(* CoDeSys 2.3 library: TcDrive.lib *)
(* Libraries: STANDARD.LIB 5.6.98 12:03:02, TcBase.lib 14.5.09 12:14:08, TcSystem.lib*7.6.16 10:01:20, TcUtilities.lib*3.2.16 15:08:58, TcEtherCAT.lib*30.11.16 15:34:02, TcTestAndSet.lib 23.2.09 12:50:08 *)

(* Global variable list: Global_Variables *)
VAR_GLOBAL CONSTANT
	S_0_IDN		: WORD	:= 16#0000;
	S_1_IDN		: WORD	:= 16#1000;
	S_2_IDN		: WORD	:= 16#2000;
	S_3_IDN		: WORD	:= 16#3000;
	S_4_IDN		: WORD	:= 16#4000;
	S_5_IDN		: WORD	:= 16#5000;
	S_6_IDN		: WORD	:= 16#6000;
	S_7_IDN		: WORD	:= 16#7000;

	P_0_IDN		: WORD	:= 16#8000;
	P_1_IDN		: WORD	:= 16#9000;
	P_2_IDN		: WORD	:= 16#A000;
	P_3_IDN		: WORD	:= 16#B000;
	P_4_IDN		: WORD	:= 16#C000;
	P_5_IDN		: WORD	:= 16#D000;
	P_6_IDN		: WORD	:= 16#E000;
	P_7_IDN		: WORD	:= 16#F000;
END_VAR
{library private}
VAR_GLOBAL CONSTANT
	iMaxNumOfDrivesUpdate 	: INT := 255;
END_VAR
VAR_GLOBAL
	bBlockEcatScan	 		: BOOL;
	iBlockEcatScanCount		: DINT;
	bBlockDrivesFwUpdate	: BOOL;
	iArrDrivesUpdatePorts 	: ARRAY [0..iMaxNumOfDrivesUpdate] OF UINT;
END_VAR

(* Data type *)
TYPE E_AX5000_DriveOpMode : (
	eOPM_NoModeOfOperation 	:= 0,
	eOPM_TorqueCtrl			:= 1,
	eOPM_VeloCtrl 			:= 2,
	eOPM_PosCtrlFbk1 		:= 3,
	eOPM_PosCtrlFbk2 		:= 4,
	eOPM_PosCtrlFbk1LagLess := 11,
	eOPM_PosCtrlFbk2LagLess := 12
);
END_TYPE

(* Data type *)
TYPE E_FwUpdateState : (
	(* update states *)
	eFwU_NoError := 0,
	eFwU_CheckCfgIdentity,
	eFwU_CheckSlaveCount,
	eFwU_CheckFindSlavePos,
	eFwU_WaitForScan,
	eFwU_ScanningSlaves,
	eFwU_CheckScannedIdentity,
	eFwU_CheckScannedFirmware,
	eFwU_FindFirmwareFile,
	eFwU_WaitForUpdate,
	eFwU_WaitForSlaveState,
	eFwU_StartFwUpdate,
	eFwU_FwUpdateInProgress,
	eFwU_FwUpdateDone,
	eFwU_NoFwUpdateRequired,

	(* not updating via this channel *)
	eFwU_UpdateViaOtherChannelActive,
	eFwU_UpdatedViaOtherChannel,

	(* error states *)
	eFwU_GetSlaveIdentityError			:= -1,
	eFwU_GetSlaveCountError				:= -2,
	eFwU_GetSlaveAddrError				:= -3,
	eFwU_StartScanError					:= -4,
	eFwU_ScanStateError					:= -5,
	eFwU_ScanIdentityError				:= -6,
	eFwU_GetSlaveStateError				:= -7,
	eFwU_ScanFirmwareError				:= -8,
	eFwU_FindFileError					:= -9,
	eFwU_CfgTypeInNoAX5xxx				:= -10,
	eFwU_ScannedTypeInNoAX5xxx			:= -11,
	eFwU_ChannelMismatch				:= -12,
	eFwU_ChannelMismatch_1Cfg_2Scanned	:= -13,
	eFwU_ChannelMismatch_2Cfg_1Scanned	:= -14,
	eFwU_CurrentMismatch				:= -15,
	eFwU_FwUpdateError					:= -16,
	eFwU_ReqSlaveStateError				:= -17,
	eFwU_ChannelMismatch_0Cfg_1Scanned	:= -18,
	eFwU_ChannelMismatch_0Cfg_2Scanned	:= -19,
	eFwU_ChannelMismatch_1Cfg_0Scanned	:= -20,
	eFwU_ChannelMismatch_2Cfg_0Scanned	:= -21,
	eFwU_TypeIncompatibleCfgToScanned	:= -22
);
END_TYPE

(* Data type *)
TYPE E_IndraDriveCs_DriveOpMode : (
	eIDC_NoModeOfOperation := 0,
	eIDC_TorqueCtrl		:= 1,
	eIDC_VeloCtrl 			:= 2,

	eIDC_PosCtrlFbk1 		:= 3,
	eIDC_PosCtrlFbk2 		:= 4,
	eIDC_PosCtrlFbk1LagLess := 11,
	eIDC_PosCtrlFbk2LagLess := 12,

	eIDC_DrvInternInterpolFbk1 := 19,
	eIDC_DrvInternInterpolFbk2 := 20,
	eIDC_DrvInternInterpolFbk1LagLess := 27,
	eIDC_DrvInternInterpolFbk2LagLess := 28,

	eIDC_PosBlockModeFbk1 := 51,
	eIDC_PosBlockModeFbk2 := 52,
	eIDC_PosBlockModeFbk1LagLess := 59,
	eIDC_PosBlockModeFbk2LagLess := 60,

	eIDC_PosCtrlDrvCtrldFbk1 := 259,
	eIDC_PosCtrlDrvCtrldFbk2 := 260,
	eIDC_PosCtrlDrvCtrldFbk1LagLess := 267,
	eIDC_PosCtrlDrvCtrldFbk2LagLess := 268,

	eIDC_DrvCtrldPositioningFbk1 := 531,
	eIDC_DrvCtrldPositioningFbk2 := 532,
	eIDC_DrvCtrldPositioningFbk1LagLess := 539,
	eIDC_DrvCtrldPositioningFbk2LagLess := 540,

	eIDC_CamFbk1VirtMaster := -30717,
	eIDC_CamFbk2VirtMaster := -30716,
	eIDC_CamFbk1VirtMasterLagLess := -30709,
	eIDC_CamFbk2VirtMasterLagLess := -30708,

	eIDC_CamFbk1RealMaster := -30701,
	eIDC_CamFbk2RealMaster := -30700,
	eIDC_CamFbk1RealMasterLagLess := -30693,
	eIDC_CamFbk2RealMasterLagLess := -30692,

	eIDC_PhaseSyncFbk1VirtMaster := -28669,
	eIDC_PhaseSyncFbk2VirtMaster := -28668,
	eIDC_PhaseSyncFbk1VirtMasterLagLess := -28661,
	eIDC_PhaseSyncFbk2VirtMasterLagLess := -28660,

	eIDC_PhaseSyncFbk1RealMaster := -28653,
	eIDC_PhaseSyncFbk2RealMaster := -28652,
	eIDC_PhaseSyncFbk1RealMasterLagLess := -28645,
	eIDC_PhaseSyncFbk2RealMasterLagLess := -28644,

	eIDC_VeloSyncVirtMaster := -24574,
	eIDC_VeloSyncRealMaster := -24558,

	eIDC_MotionProfileFbk1VirtMaster := -26621,
	eIDC_MotionProfileFbk2VirtMaster := -26620,
	eIDC_MotionProfileLagLessFbk1VirtMaster := -26613,
	eIDC_MotionProfileLagLessFbk2VirtMaster := -26612,

	eIDC_MotionProfileFbk1RealMaster := -26605,
	eIDC_MotionProfileFbk2RealMaster := -26604,
	eIDC_MotionProfileLagLessFbk1RealMaster := -26597,
	eIDC_MotionProfileLagLessFbk2RealMaster := -26596,

	eIDC_PosCtrlDrvCtrld := 773,
	eIDC_DrvCtrldPositioning := 533,
	eIDC_PosBlockMode := 565,
	eIDC_VeloSynchronization := 66,
	eIDC_PosSynchronization := 581

);
END_TYPE

(* Data type *)
TYPE E_SoE_AttribLen : (
	eSoE_LEN_2BYTE	:= 1,
	eSoE_LEN_4BYTE	:= 2,
	eSoE_LEN_8BYTE	:= 3,
	eSoE_LEN_V1BYTE	:= 4,
	eSoE_LEN_V2BYTE	:= 5,
	eSoE_LEN_V4BYTE	:= 6,
	eSoE_LEN_V8BYTE	:= 7
);
END_TYPE

(* Data type *)
TYPE E_SoE_CmdControl :(
	eSoE_CmdControl_Cancel				:= 0,
	eSoE_CmdControl_Set					:= 1,
	eSoE_CmdControl_SetAndEnable		:= 3
	);
END_TYPE

(* Data type *)
TYPE E_SoE_CmdState :(
	eSoE_CmdState_NotSet					:= 0,
	eSoE_CmdState_Set						:= 1,
	eSoE_CmdState_Executed					:= 2,
	eSoE_CmdState_SetEnabledExecuted		:= 3,
	eSoE_CmdState_SetAndInterrupted			:= 5,
	eSoE_CmdState_SetEnabledNotExecuted	:= 7,
	eSoE_CmdState_Error						:= 15
);
END_TYPE

(* Data type *)
TYPE E_SoE_Type : (
	eSoE_Type_BIN			:= 0,
	eSoE_Type_UNSIGNED	:= 1,
	eSoE_Type_SIGNED		:= 2,
	eSoE_Type_HEX			:= 3,
	eSoE_Type_TEXT		:= 4,
	eSoE_Type_IDN			:= 5,
	eSoE_Type_FLOAT		:= 6
);
END_TYPE

(* Data type *)
TYPE ST_AX5000_C1D :
STRUCT
	bOverloadShutdown			: BOOL; (* C1D Bit  0 *)
	bAmplifierOverTempShutdown	: BOOL; (* C1D Bit  1 *)
	bMotorOverTempShutdown		: BOOL; (* C1D Bit  2 *)
	bCoolingErrorShutdown		: BOOL; (* C1D Bit  3 *)

	bControlVoltageError		: BOOL; (* C1D Bit  4 *)
	bFeedbackError				: BOOL; (* C1D Bit  5 *)
	bCommunicationError			: BOOL; (* C1D Bit  6 *)
	bOverCurrentError			: BOOL; (* C1D Bit  7 *)

	bOverVoltageError			: BOOL; (* C1D Bit  8 *)
	bUnderVoltageError			: BOOL; (* C1D Bit  9 *)
	bPowerSupplyPhaseError		: BOOL; (* C1D Bit 10 *)
	bExcessivePosDiviationError : BOOL; (* C1D Bit 11 *)

	bCommunicationErrorBit		: BOOL; (* C1D Bit 12 *)
	bOvertravelLimitExceeeded	: BOOL; (* C1D Bit 13 *)
	bReserved 					: BOOL; (* C1D Bit 14 *)
	bManufacturerSpecificError	: BOOL; (* C1D Bit 15 *)
END_STRUCT
END_TYPE

(* Data type *)
TYPE ST_AX5000DriveStatus :
STRUCT
	bStatusCmdValProcessing 	: BOOL;
	bRealTimeStatusBit1 		: BOOL;
	bRealTimeStatusBit2 		: BOOL;
	bDrvShutdownBitC1D		 	: BOOL;
	bChangeBitC2D		 		: BOOL;
	bChangeBitC3D		 		: BOOL;
	bNotReadyToPowerUp			: BOOL;
	bReadyForPower				: BOOL;
	bReadyForEnable				: BOOL;
	bEnabled					: BOOL;
	iActOpModeParNum			: UINT;
	eActOpMode					: E_AX5000_DriveOpMode;
	iReserved					: UINT;
END_STRUCT
END_TYPE

(* Data type *)
TYPE ST_IndraDriveCs_C1D :
STRUCT
	bOverloadShutdown			: BOOL; (* C1D Bit  0 *)
	bAmplifierOverTempShutdown	: BOOL; (* C1D Bit  1 *)
	bMotorOverTempShutdown		: BOOL; (* C1D Bit  2 *)
	bReserved_3					: BOOL; (* C1D Bit  3 *)

	bControlVoltageError		: BOOL; (* C1D Bit  4 *)
	bFeedbackError				: BOOL; (* C1D Bit  5 *)
	bReserved_6					: BOOL; (* C1D Bit  6 *)
	bOverCurrentError			: BOOL; (* C1D Bit  7 *)

	bOverVoltageError			: BOOL; (* C1D Bit  8 *)
	bUnderVoltageError			: BOOL; (* C1D Bit  9 *)
	bReserved_10				: BOOL; (* C1D Bit 10 *)
	bExcessivePosDiviationError : BOOL; (* C1D Bit 11 *)

	bCommunicationErrorBit		: BOOL; (* C1D Bit 12 *)
	bOvertravelLimitExceeeded	: BOOL; (* C1D Bit 13 *)
	bReserved_14				: BOOL; (* C1D Bit 14 *)
	bManufacturerSpecificError	: BOOL; (* C1D Bit 15 *)
END_STRUCT
END_TYPE

(* Data type *)
TYPE ST_IndraDriveCsDriveStatus :
STRUCT
	bStatusCmdValProcessing 	: BOOL;
	bRealTimeStatusBit1 		: BOOL;
	bRealTimeStatusBit2 		: BOOL;
	bDrvShutdownBitC1D		 	: BOOL;
	bChangeBitC2D		 		: BOOL;
	bChangeBitC3D		 		: BOOL;
	bNotReadyToPowerUp			: BOOL;
	bReadyForPower				: BOOL;
	bReadyForEnable				: BOOL;
	bEnabled					: BOOL;
	iActOpModeParNum			: UINT;
	eActOpMode					: E_IndraDriveCs_DriveOpMode;
	iReserved					: UINT;
END_STRUCT
END_TYPE

(* Data type *)
TYPE ST_SoE_CPxInvParamList : ST_SoE_CPxInvParamList25;
END_TYPE

(* Data type *)
TYPE ST_SoE_CPxInvParamList25 :
STRUCT
	iActualSize 	: UINT;
	iMaxSize 		: UINT;
	arrIdnNumbers	: ARRAY [1..25] OF UDINT;
END_STRUCT
END_TYPE

(* Data type *)
TYPE ST_SoE_DiagNumList : ST_SoE_DiagNumList30;
END_TYPE

(* Data type *)
TYPE ST_SoE_DiagNumList30 :
STRUCT
	iActualSize 	: UINT;
	iMaxSize 		: UINT;
	arrDiagNumbers	: ARRAY [0..29] OF UDINT;
END_STRUCT
END_TYPE

(* Data type *)
TYPE ST_SoE_DiagNumList50 :
STRUCT
	iActualSize 	: UINT;
	iMaxSize 		: UINT;
	arrDiagNumbers	: ARRAY [0..49] OF UDINT;
END_STRUCT
END_TYPE

(* Data type *)
TYPE ST_SoE_String :
STRUCT
	iActualSize : UINT;
	iMaxSize 	: UINT;
	strData		: STRING(MAX_STRING_LENGTH);
END_STRUCT
END_TYPE

(* Data type *)
TYPE ST_SoE_StringEx :
STRUCT
	dwAttribute : DWORD;
	iActualSize : UINT;
	iMaxSize 	: UINT;
	strData		: STRING(MAX_STRING_LENGTH);
END_STRUCT
END_TYPE

(* POU F_ConvWordToSTAX5000C1D, ST *)
FUNCTION F_ConvWordToSTAX5000C1D : ST_AX5000_C1D
VAR_INPUT
	wClass1Diag  : WORD;
END_VAR
VAR
	stAX5000C1D	: ST_AX5000_C1D;
END_VAR
stAX5000C1D.bOverloadShutdown			:= wClass1Diag.0;
stAX5000C1D.bAmplifierOverTempShutdown	:= wClass1Diag.1;
stAX5000C1D.bMotorOverTempShutdown		:= wClass1Diag.2;
stAX5000C1D.bCoolingErrorShutdown		:= wClass1Diag.3;

stAX5000C1D.bControlVoltageError		:= wClass1Diag.4;
stAX5000C1D.bFeedbackError				:= wClass1Diag.5;
stAX5000C1D.bCommunicationError			:= wClass1Diag.6;
stAX5000C1D.bOverCurrentError			:= wClass1Diag.7;

stAX5000C1D.bOverVoltageError			:= wClass1Diag.8;
stAX5000C1D.bUnderVoltageError			:= wClass1Diag.9;
stAX5000C1D.bPowerSupplyPhaseError		:= wClass1Diag.10;
stAX5000C1D.bExcessivePosDiviationError := wClass1Diag.11;

stAX5000C1D.bCommunicationErrorBit		:= wClass1Diag.12;
stAX5000C1D.bOvertravelLimitExceeeded	:= wClass1Diag.13;
stAX5000C1D.bReserved 					:= wClass1Diag.14;
stAX5000C1D.bManufacturerSpecificError	:= wClass1Diag.15;

F_ConvWordToSTAX5000C1D := stAX5000C1D;
END_FUNCTION

(* POU F_ConvWordToSTAX5000DriveStatus, ST *)
FUNCTION F_ConvWordToSTAX5000DriveStatus : ST_AX5000DriveStatus
VAR_INPUT
	wDriveStatus  	: WORD;
END_VAR
VAR
	stDriveStatus	: ST_AX5000DriveStatus;
	iOpModeSelect	: INT;
END_VAR
stDriveStatus.bStatusCmdValProcessing := wDriveStatus.3;

stDriveStatus.bRealTimeStatusBit1 := wDriveStatus.6;
stDriveStatus.bRealTimeStatusBit2 := wDriveStatus.7;

iOpModeSelect := 0;
IF wDriveStatus.8 THEN
	iOpModeSelect := iOpModeSelect + 1;
END_IF
IF wDriveStatus.9 THEN
	iOpModeSelect := iOpModeSelect + 2;
END_IF
IF wDriveStatus.10 THEN
	iOpModeSelect := iOpModeSelect + 4;
END_IF

CASE iOpModeSelect OF
0: stDriveStatus.iActOpModeParNum := 32;
1: stDriveStatus.iActOpModeParNum := 33;
2: stDriveStatus.iActOpModeParNum := 34;
3: stDriveStatus.iActOpModeParNum := 35;
4: stDriveStatus.iActOpModeParNum := 284;
5: stDriveStatus.iActOpModeParNum := 285;
6: stDriveStatus.iActOpModeParNum := 286;
7: stDriveStatus.iActOpModeParNum := 287;
END_CASE

stDriveStatus.bChangeBitC3D			:= wDriveStatus.11;
stDriveStatus.bChangeBitC2D			:= wDriveStatus.12;
stDriveStatus.bDrvShutdownBitC1D	:= wDriveStatus.13;

IF wDriveStatus.14 THEN
	IF wDriveStatus.15 THEN (* 3 *)
		stDriveStatus.bNotReadyToPowerUp := FALSE;
		stDriveStatus.bReadyForPower := TRUE;
		stDriveStatus.bReadyForEnable := TRUE;
		stDriveStatus.bEnabled := TRUE;
	ELSE (* 1 *)
		stDriveStatus.bNotReadyToPowerUp := FALSE;
		stDriveStatus.bReadyForPower := TRUE;
		stDriveStatus.bReadyForEnable := FALSE;
		stDriveStatus.bEnabled := FALSE;
	END_IF
ELSE
	IF wDriveStatus.15 THEN (* 2 *)
		stDriveStatus.bNotReadyToPowerUp := FALSE;
		stDriveStatus.bReadyForPower := TRUE;
		stDriveStatus.bReadyForEnable := TRUE;
		stDriveStatus.bEnabled := FALSE;
	ELSE (* 0 *)
		stDriveStatus.bNotReadyToPowerUp := TRUE;
		stDriveStatus.bReadyForPower := FALSE;
		stDriveStatus.bReadyForEnable := FALSE;
		stDriveStatus.bEnabled := FALSE;
	END_IF
END_IF
F_ConvWordToSTAX5000DriveStatus := stDriveStatus;
END_FUNCTION

(* POU F_ConvWordToSTIndraDriveCsC1D, ST *)
FUNCTION F_ConvWordToSTIndraDriveCsC1D : ST_IndraDriveCs_C1D
VAR_INPUT
	wClass1Diag  : WORD;
END_VAR
VAR
	stIndraDriveCsC1D	: ST_IndraDriveCs_C1D;
END_VAR
stIndraDriveCsC1D.bOverloadShutdown				:= wClass1Diag.0;
stIndraDriveCsC1D.bAmplifierOverTempShutdown	:= wClass1Diag.1;
stIndraDriveCsC1D.bMotorOverTempShutdown		:= wClass1Diag.2;
stIndraDriveCsC1D.bReserved_3					:= wClass1Diag.3;

stIndraDriveCsC1D.bControlVoltageError			:= wClass1Diag.4;
stIndraDriveCsC1D.bFeedbackError				:= wClass1Diag.5;
stIndraDriveCsC1D.bReserved_6					:= wClass1Diag.6;
stIndraDriveCsC1D.bOverCurrentError				:= wClass1Diag.7;

stIndraDriveCsC1D.bOverVoltageError				:= wClass1Diag.8;
stIndraDriveCsC1D.bUnderVoltageError			:= wClass1Diag.9;
stIndraDriveCsC1D.bReserved_10					:= wClass1Diag.10;
stIndraDriveCsC1D.bExcessivePosDiviationError 	:= wClass1Diag.11;

stIndraDriveCsC1D.bCommunicationErrorBit		:= wClass1Diag.12;
stIndraDriveCsC1D.bOvertravelLimitExceeeded		:= wClass1Diag.13;
stIndraDriveCsC1D.bReserved_14 					:= wClass1Diag.14;
stIndraDriveCsC1D.bManufacturerSpecificError	:= wClass1Diag.15;

F_ConvWordToSTIndraDriveCsC1D := stIndraDriveCsC1D;
END_FUNCTION

(* POU F_ConvWordToSTIndraDriveCsDriveStatus, ST *)
FUNCTION F_ConvWordToSTIndraDriveCsDriveStatus : ST_IndraDriveCsDriveStatus
VAR_INPUT
	wDriveStatus  	: WORD;
END_VAR
VAR
	stDriveStatus	: ST_IndraDriveCsDriveStatus;
	iOpModeSelect	: INT;
END_VAR
stDriveStatus.bStatusCmdValProcessing := wDriveStatus.3;

stDriveStatus.bRealTimeStatusBit1 := wDriveStatus.6;
stDriveStatus.bRealTimeStatusBit2 := wDriveStatus.7;

iOpModeSelect := 0;
IF wDriveStatus.8 THEN
	iOpModeSelect := iOpModeSelect + 1;
END_IF
IF wDriveStatus.9 THEN
	iOpModeSelect := iOpModeSelect + 2;
END_IF
IF wDriveStatus.10 THEN
	iOpModeSelect := iOpModeSelect + 4;
END_IF

CASE iOpModeSelect OF
0: stDriveStatus.iActOpModeParNum := 32;
1: stDriveStatus.iActOpModeParNum := 33;
2: stDriveStatus.iActOpModeParNum := 34;
3: stDriveStatus.iActOpModeParNum := 35;
4: stDriveStatus.iActOpModeParNum := 284;
5: stDriveStatus.iActOpModeParNum := 285;
6: stDriveStatus.iActOpModeParNum := 286;
7: stDriveStatus.iActOpModeParNum := 287;
END_CASE

stDriveStatus.bChangeBitC3D			:= wDriveStatus.11;
stDriveStatus.bChangeBitC2D			:= wDriveStatus.12;
stDriveStatus.bDrvShutdownBitC1D	:= wDriveStatus.13;

IF wDriveStatus.14 THEN
	IF wDriveStatus.15 THEN (* 3 = AF *)
		stDriveStatus.bNotReadyToPowerUp := FALSE;
		stDriveStatus.bReadyForPower := TRUE;
		stDriveStatus.bReadyForEnable := TRUE;
		stDriveStatus.bEnabled := TRUE;
	ELSE (* 1 = bb *)
		stDriveStatus.bNotReadyToPowerUp := FALSE;
		stDriveStatus.bReadyForPower := TRUE;
		stDriveStatus.bReadyForEnable := FALSE;
		stDriveStatus.bEnabled := FALSE;
	END_IF
ELSE
	IF wDriveStatus.15 THEN (* 2 = AB *)
		stDriveStatus.bNotReadyToPowerUp := FALSE;
		stDriveStatus.bReadyForPower := TRUE;
		stDriveStatus.bReadyForEnable := TRUE;
		stDriveStatus.bEnabled := FALSE;
	ELSE (* 0 = e.g. P2 *)
		stDriveStatus.bNotReadyToPowerUp := TRUE;
		stDriveStatus.bReadyForPower := FALSE;
		stDriveStatus.bReadyForEnable := FALSE;
		stDriveStatus.bEnabled := FALSE;
	END_IF
END_IF
F_ConvWordToSTIndraDriveCsDriveStatus := stDriveStatus;
END_FUNCTION

(* POU F_GetVersionTcDrive, ST *)
FUNCTION F_GetVersionTcDrive : UINT
(* Returns the library version information  *)
VAR_INPUT
	nVersionElement       :       INT;
END_VAR
VAR
END_VAR
(* Version history:
Date          	| Version 	| created under 	     	| Author	| Remark 
------------------------------------------------------------------------------------------------------------------------------------------------------ 
15.05.2008    	| 0.0.1     | V2.10.0 (Build 1325) 		| I.Ch.		| first release 
13.06.2008    	| 0.0.2     | V2.10.0 (Build 1325) 		| I.Ch.		| FB_SoEAX5000Reset_ByDriveRef added
17.06.2008		| 0.0.3		| V2.10.0 (Build 1326)		| AnK		| Don't read the attribute from P-0-0352 in FB_SoEAX5000Reset_ByDriveRef
10.07.2008		| 0.0.4		| V2.10.0 (Build 1326)		| PKa		| FB_SoEAX5000Reset_ByDriveRef, Reset sequence changed PreOP-S.0.0099-OP
11.07.2008		| 0.0.5		| V2.10.0 (Build 1328)		| PKa		| FB_SoEAX5000Reset_ByDriveRef, Read S.0.0011 for DriveError, Reset sequence changed S.0.0099-ClearErrorOP
28.07.2008		| 0.0.6		| V2.10.0 (Build 1328)		| I.Ch.		| using of ST_DriveRef instead of ST_SoE_DriveRef
28.08.2008		| 0.0.7		| V2.10.0 (Build 1328)		| I.Ch.		| FB_SoEAX5000Reset_ByDriveRef removed, FB_SoEReset_ByDriveRef modified
29.09.2008		| 0.0.8		| V2.10.0 (Build 1328)		| I.Ch.		| FB_SoEReset_ByDriveRef: removed check for OP state
02.10.2008		| 0.0.9		| V2.10.0 (Build 1328)		| I.Ch.		| folders added
12.12.2008		| 0.0.10	| V2.10.0 (Build 1330)		| I.Ch.		| FB_SoEAX5000FirmwareUpdate_ByDriveRef added
12.12.2008		| 0.0.11	| V2.10.0 (Build 1330)		| I.Ch.		| TestAndSet semaphore added
13.12.2008		| 0.0.12	| V2.10.0 (Build 1330)		| I.Ch.		| parallel firmware download added
15.12.2008		| 0.0.13	| V2.10.0 (Build 1330)		| I.Ch.		| cleanup
16.12.2008		| 0.0.14	| V2.10.0 (Build 1330)		| I.Ch.		| provide FB_EcFoeLoad.sInfo as iDiagNumber
16.01.2009		| 0.0.15	| V2.10.0 (Build 1331)		| I.Ch.		| provide FirmwareUpdate for >128 EtherCAT Slaves
22.01.2009		| 0.0.16	| V2.11.0 (Build 1513)		| AnK		| FB_SoEAX5000FirmwareUpdate_ByDriveRef: Change file names from AX5200-0000- to AX52xx-xxxx-
03.02.2009		| 0.0.17	| V2.11.0 (Build 1332)		| I.Ch.		| FB_SoEAX5000FirmwareUpdate_ByDriveRef: Change file names AX51/AX52xx-xxxx- to AX5yxx-xxxx-; added AX50**-xxxx
04.02.2009		| 0.0.18	| V2.11.0 (Build 1332)		| I.Ch.		| FB_SoEAX5000FirmwareUpdate_ByDriveRef: fix for filename: '_' instead of '-' (AX5yxx_xxxx_...) 
05.02.2009		| 0.0.19	| V2.11.0 (Build 1332)		| I.Ch.		| cleanup 
15.03.2009		| 0.0.20	| V2.11.0 (Build 1334)		| I.Ch.		| FB_SoEReadClassXDiag_ByDriveRef added, reads C1D|C2D|C3D class diag, F_ConvWordToSTAX5000C1D + ST_AX5000_C1D added 
19.03.2009		| 0.0.21	| V2.11.0 (Build 1334)		| I.Ch.		| Conversion FUs for DriveState/EcSlaveState + DTs DriveState/EcSlaveState, ST_SoE_CPxInvParamList added 
23.03.2009		| 0.0.22	| V2.11.0 (Build 1334)		| I.Ch.		| Conversion FUs for EcSlaveState + EcSlaveState move to TcEtherCAT.lib added 
19.10.2009		| 0.0.23	| V2.11.0 (Build 1539)		| I.Ch.		| optional sequential reading of attribute and value (bSeqReadDrvAttrAndValue) added for other drives than AX5000 in
																		FB_SoEReadClassXDiag_ByDriveRef, FB_SoEReadDiagMessage_ByDriveRef, FB_SoEReadDiagNumber_ByDriveRef, FB_SoEReadAmplifierTemperature_ByDriveRef
																		FB_SoEReadDcBusCurrent_ByDriveRef, FB_SoEReadDcBusVoltage_ByDriveRef, FB_SoEReadMotorTemperature_ByDriveRef
19.10.2009		| 0.0.24	| V2.11.0 (Build 1539)		| I.Ch.		| bSeqReadDrvAttrAndValue moved to TcEtherCAT.lib
13.01.2010		| 0.0.25	| V2.11.0 (Build 1541)		| I.Ch.		| ST_SoE_DiagNumList30, ST_SoE_DiagNumList50 added, ST_SoE_DiagNumList as ALIAS type; ST_SoE_CPxInvParamList25 added, ST_SoE_CPxInvParamList as ALIAS type 
																		Conversion Functions/Datatypes for IndraDriveCs added
17.03.2010		| 0.0.26	| V2.11.0 (Build 1544)		| AnK.		| FB_SoEExecuteCommand_ByDriveRef: Change the handling in case of a command error
02.10.2012		| 0.0.27	| V2.11.0 (Build 1557)		| I.Ch.		| FB_SoEAX5000FirmwareUpdate_ByDriveRef supports FW Update for HW2 in compatible mode (HW1 configured)
24.01.2017		| 0.0.28	| V2.11.0 (Build 2256)		| I.Ch.		| FB_SoEAX5000FirmwareUpdate_ByDriveRef adjusted to also use "_dual_use_conform" firmware files
*)
CASE nVersionElement OF
1: (* major number *)
       F_GetVersionTcDrive := 0;
2: (* minor number *)
       F_GetVersionTcDrive := 0;
3: (* revision number *)
       F_GetVersionTcDrive := 28;
ELSE
   F_GetVersionTcDrive := 16#FFFF;
END_CASE
END_FUNCTION

(* POU FB_SoEAX5000FirmwareUpdate_ByDriveRef, ST *)
FUNCTION_BLOCK FB_SoEAX5000FirmwareUpdate_ByDriveRef
VAR_INPUT
	stDriveRef				: ST_DriveRef; 	(* contains sNetID of EcMaster, nSlaveAddr of EcDrive, nDriveNo of EcDrive, either preset or read from NC *)
	bExecute				: BOOL;			(* Function block execution is triggered by a rising edge at this input.*)
	tTimeout				: TIME := DEFAULT_ADS_TIMEOUT;(* States the time before the function is cancelled. *)
	sFirmwareVersion		: STRING(20);	(* version string vx_yy_bnnnn,
												"v1.05_b0009" 		for specific build: v1.05 Build 0009, 
												"v1.05_b00??" 		for specific version v1.05 latest release build, 
												"v1.??_b00??" 		for latest v1.xx version latest release build
												"v?.??_b00??", "" 	for latest version latest release build 

												"v1.05_b10??" - "v1_05_b89??"  	
																	for specific version v1.05 latest customer specific build, 
												"v1.05_b90??" 		for specific version v1.05 latest debug build, 

												same wildcards for versions 2.xx Build yyyy
												"v2.03_b0026" 		for specific build: v2.03 Build 0026, 
												"v2.03_b00??" 		for specific version v2.03 latest release build, 
												...
											*)
	sFirmwarePath			: T_MaxString;	(* drive:\path, e.g. "C:\TwinCAT\Io\TcDriveManager\FirmwarePool" *)
	sNetIdIPC				: T_AmsNetId;
	iReqEcState				: UINT := EC_DEVICE_STATE_OP;
END_VAR
VAR_OUTPUT
	bBusy					: BOOL;
	bError					: BOOL;
	iAdsErrId				: UINT;
	iSercosErrId			: UINT;
	iDiagNumber				: UDINT;
	eFwUpdateState			: E_FwUpdateState;
	iLoadProgress			: INT;
	sSelectedFirmwareFile	: STRING(MAX_STRING_LENGTH);	(* found firmware file, e.g. "AX5yxx_xxxx_0010_v1_05_b0009.efw" or "AX5yxx_xxxx_0010_v1_05_b0009_dual_use_conform.efw" *)
END_VAR
{library private}
VAR
	iState					: INT;
	bExecute_I				: BOOL;
	iErrId					: UDINT;
	I						: DINT;
	iNextUpdateIdx			: INT;
	iCurUpdateIdx			: INT;
	bUpdateViaOtherChn		: BOOL;

	sConfiguredType 		: STRING(20);	(* type of slave, e.g. "AX5206-0000-0009" *)
	sScannedType 			: STRING(20);	(* type of slave, e.g. "AX5206-0000-0010" *)

	sConfiguredFirmwareFile		: STRING(MAX_STRING_LENGTH);(* configured firmware file, e.g. 	"AX5yxx_xxxx_0010_v1_05_b0003.efw" or "AX5021_xxxx_0009_v1_04_b0002.efw" *)
	sScannedFirmwareFile		: STRING(MAX_STRING_LENGTH);(* scanned firmware file, e.g. 		"AX5yxx_xxxx_0010_v1_05_b0003.efw" or "AX5021_xxxx_0009_v1_04_b0002.efw" *)
	sCompatibleFirmwareFile		: STRING(MAX_STRING_LENGTH);(* compatible firmware file, e.g. 	"AX5yxx_xxxx_0200_v2_03_b0026.efw" or "AX5021_xxxx_0200_v2_03_b0026.efw" *)

	sConfiguredFirmwareFileDUC	: STRING(MAX_STRING_LENGTH);(* configured firmware file, e.g. 	"AX5yxx_xxxx_0010_v1_05_b0003_dual_use_conform.efw" or "AX5021_xxxx_0009_v1_04_b0002_dual_use_conform.efw" *)
	sScannedFirmwareFileDUC		: STRING(MAX_STRING_LENGTH);(* scanned firmware file, e.g. 		"AX5yxx_xxxx_0010_v1_05_b0003_dual_use_conform.efw" or "AX5021_xxxx_0009_v1_04_b0002_dual_use_conform.efw" *)
	sCompatibleFirmwareFileDUC	: STRING(MAX_STRING_LENGTH);(* compatible firmware file, e.g. 	"AX5yxx_xxxx_0200_v2_03_b0026_dual_use_conform.efw" or "AX5021_xxxx_0200_v2_03_b0026_dual_use_conform.efw" *)
	sSelectedFirmwareFileDUC	: STRING(MAX_STRING_LENGTH);(* found firmware file, e.g. 		"AX5yxx_xxxx_0010_v1_05_b0009_dual_use_conform.efw" *)

	(* 1. *)
	fbEcGetSlaveIdentity	: FB_EcGetSlaveIdentity;
	stIdentity				: ST_EcSlaveIdentity;	(*Slave identity of the EtherCAT slave devie.*)

	(* 2. *)
	fbEcGetSlaveCount		: FB_EcGetSlaveCount;
	nTotalSlaves			: UINT;

	(* 3. *)
	fbAdsRead				: ADSREAD;
	nSlavesRead				: UINT;
	nBlockIndex 			: UINT;
	nSlaves					: UINT;

	(* 4. *)
	fbCoERead				: FB_EcCoESdoReadEx;
	nSlaveArr				: ARRAY [0..128] OF UINT;
	iSlaveIndex				: UINT;
	iSlaveBlockIndex		: UINT;
	bPositionFound 			: BOOL;

	(* 6. *)
	fbAdsWrite				: ADSWRITE;
	stScanStatus			: ST_EcScannedSlaveStatus;
	nIdxOffs				: UDINT;
	nScanCommand 			: WORD := 16#FFFF;
	stLocalInfo				: ST_EcSlaveScannedData;

	(* 9. *)
	fbEcGetSlaveState		: FB_EcGetSlaveState;
	iSlaveState				: WORD;

	(* 10. *)
	fbGetSwSoE				: FB_SoERead_ByDriveRef;
	stSoEValue				: ST_SoE_String;
	sScannedFirmwareVersion : STRING(80);	(* scanned firmware version, e.g. "Firmware: v1.05 (Build 0009) / Bootloader: v1.02 (Build 0001)" *)
	sScannedVBString		: STRING(20);	(* extracted from scanned firmware version, e.g. v1_05_b0009 *)
	sTemp					: STRING(20);
	iStrPosV				: INT;
	iStrPosDot				: INT;
	iStrPosBuild			: INT;

	(* 11. *)
	fbFindFiles				: FB_EnumFindFileEntry;
	stFindFile				: ST_FindFileEntry; (* Find file entry *)
	eCmd					: E_EnumCmdType	:= eEnumCmd_First; (* Enumerator navigation command *)
	bNoMoreFiles			: BOOL;
	sFoundFirmwareFile	 	: STRING(MAX_STRING_LENGTH);	(* found firmware file, e.g. "AX5yxx_xxxx_0010_v1_05_b0003.efw" *)
	iFilesFound				: UDINT;
	bExecFind				: BOOL;

	fbFindFilesDUC			: FB_EnumFindFileEntry;
	stFindFileDUC			: ST_FindFileEntry; (* Find file entry *)
	eCmdDUC					: E_EnumCmdType	:= eEnumCmd_First; (* Enumerator navigation command *)
	bNoMoreFilesDUC			: BOOL;
	sFoundFirmwareFileDUC 	: STRING(MAX_STRING_LENGTH);	(* found firmware file, e.g. "AX5yxx_xxxx_0010_v1_05_b0003.efw" *)
	iFilesFoundDUC			: UDINT;
	bExecFindDUC			: BOOL;

	bUseLatestBuild			: BOOL;
	bCompatibleMode			: BOOL;
	bIncompatibleType		: BOOL;

	(* 13. *)
	DelayTimer				: TON := (PT := T#3s);

	(* 14. *)
	fbEcFoeLoad				: FB_EcFoeLoad;
	sFoEInfo				: STRING(80);
	iFindStrPos				: INT;
	iByteArr4				: ARRAY [0..3] OF BYTE;

	(* 16. *)
	fbEcReqSlaveState		: FB_EcReqSlaveState;
	iNoReplyCnt: INT;
END_VAR
VAR CONSTANT
	nSDO_IDX_SBP_SLAVEINFODATASTART 	: DWORD := 16#00_00_90_00;
	nSDO_IDX_SBP_SCANCOMMANDSTART 		: DWORD := 16#00_00_F0_02;
	nSDO_IDX_SBP_SCANNEDSLAVES	 		: DWORD := 16#00_00_F0_40;
	nADSIOFFS_ECAT_COE_COMPLETEACCESS 	: DWORD := 16#00_00_01_00;
	nSDO_IDX_SBP_CONFIGUREDSLAVES	 	: DWORD := 16#00_00_F0_20;
END_VAR
CASE iState OF
0: (* idle *)
	IF bExecute AND NOT bExecute_I THEN
		bExecute_I 			:= bExecute;

		bBusy				:= TRUE;
		bError				:= FALSE;
		iErrId				:= 0;
		iAdsErrId			:= 0;
		iSercosErrId		:= 0;
		iDiagNumber			:= 0;
		nBlockIndex			:= 0;
		nSlaves				:= 0;
		nSlavesRead			:= 0;
		nTotalSlaves		:= 0;
		iLoadProgress		:= 0;
		eFwUpdateState		:= eFwU_NoError;
		bUpdateViaOtherChn 	:= FALSE;
		iState				:= iState + 1;

		(* 1. get configured revision of AX5000 *)
		fbEcGetSlaveIdentity(bExecute := FALSE);
		fbEcGetSlaveIdentity(
			sNetId		:= stDriveRef.sNetId,
			nSlaveAddr	:= stDriveRef.nSlaveAddr,
			bExecute	:= TRUE,
			tTimeout	:= tTimeout,
		);
	END_IF

1: (* wait for configured revision of AX5000 *)
	eFwUpdateState		:= eFwU_CheckCfgIdentity;

	fbEcGetSlaveIdentity();
	IF NOT fbEcGetSlaveIdentity.bBusy THEN
		IF NOT fbEcGetSlaveIdentity.bError THEN
			stIdentity 		:= fbEcGetSlaveIdentity.identity;
			sConfiguredType := F_ConvProductCodeToString(stIdentity);
			IF (LEFT(sConfiguredType, 3) <> 'AX5') THEN
				(* configured slave type <> AX5xxx *)
				eFwUpdateState := eFwU_CfgTypeInNoAX5xxx;
				bBusy		:= FALSE;
				bError		:= TRUE;
				iErrId		:= 16#70E;
				iAdsErrId	:= UDINT_TO_UINT(iErrId);
				iState		:= 0;
			ELSE
				(* create firmware file name *)
				sConfiguredFirmwareFile 	:= '';
				sConfiguredFirmwareFileDUC 	:= '';
				IF (LEFT(sConfiguredType, 4) = 'AX50') THEN
					sConfiguredFirmwareFile := LEFT(sConfiguredType, 6);								(* --> "AX5021"               *)
					sConfiguredFirmwareFile := CONCAT(sConfiguredFirmwareFile, '_xxxx_');				(* --> "AX5021_xxxx_"         *)
				ELSIF (LEFT(sConfiguredType, 4) = 'AX51') OR (LEFT(sConfiguredType, 4) = 'AX52') THEN
					sConfiguredFirmwareFile := 'AX5yxx_xxxx_';											(* --> "AX5yxx_xxxx_"         *)
				END_IF

				sConfiguredFirmwareFile := CONCAT(sConfiguredFirmwareFile, RIGHT(sConfiguredType,4));	(* --> "AX5021_xxxx_0002"           or "AX5yxx_xxxx_0009"   *)
				sConfiguredFirmwareFile := CONCAT(sConfiguredFirmwareFile, '_');						(* --> "AX5021_xxxx_0002_"          or "AX5yxx_xxxx_0009_"   *)
				IF sFirmwareVersion = '' THEN
					bUseLatestBuild := TRUE;
					sConfiguredFirmwareFile 	:= CONCAT(sConfiguredFirmwareFile, 'v?_??_b00??');			(* --> "AX5021_xxxx_0002_v?_??_b00??"        				or "AX5yxx_xxxx_0009_v?_??_b00??"  *)
					sConfiguredFirmwareFileDUC 	:= CONCAT(sConfiguredFirmwareFile, '_dual_use_conform.efw');(* --> "AX5021_xxxx_0002_v?_??_b00??_dual_use_conform.efw" 	or "AX5yxx_xxxx_0009_v?_??_b00??_dual_use_conform.efw"  *)
					sConfiguredFirmwareFile 	:= CONCAT(sConfiguredFirmwareFile, '.efw');					(* --> "AX5021_xxxx_0002_v?_??_b00??.efw" 	 				or "AX5yxx_xxxx_0009_v?_??_b00??.efw"  *)
				ELSE
					IF (FIND(sFirmwareVersion, '?') > 0) OR (FIND(sFirmwareVersion, '*') > 0) THEN
						bUseLatestBuild := TRUE;
					ELSE
						bUseLatestBuild := FALSE;
					END_IF
					iStrPosDot := FIND(sFirmwareVersion, '.');
					IF iStrPosDot > 0 THEN
						sTemp := sFirmwareVersion; 														  (* --> "v1.05_b0009" *)
						sFirmwareVersion := LEFT(sTemp, iStrPosDot-1);
						sFirmwareVersion := CONCAT(sFirmwareVersion, '_');
						sFirmwareVersion := CONCAT(sFirmwareVersion, RIGHT(sTemp, LEN(sTemp)-iStrPosDot));(* --> "v1_05_b0009" *)
					END_IF

					sConfiguredFirmwareFile 	:= CONCAT(sConfiguredFirmwareFile, sFirmwareVersion);		(* --> "AX5021_xxxx_0002_v1_05_b0009" 						or "AX5yxx_xxxx_0009_v1_05_b0009" *)
					sConfiguredFirmwareFileDUC 	:= CONCAT(sConfiguredFirmwareFile, '_dual_use_conform.efw');(* --> "AX5021_xxxx_0002_v1_05_b0009_dual_use_conform.efw" 	or "AX5yxx_xxxx_0009_v1_05_b0009_dual_use_conform.efw" *)
					sConfiguredFirmwareFile 	:= CONCAT(sConfiguredFirmwareFile, '.efw');					(* --> "AX5021_xxxx_0002_v1_05_b0009.efw" 					or "AX5yxx_xxxx_0009_v1_05_b0009.efw" *)
				END_IF
				
				sConfiguredFirmwareFile 	:= F_ToUCase(sConfiguredFirmwareFile);
				sConfiguredFirmwareFileDUC	:= F_ToUCase(sConfiguredFirmwareFileDUC);

				(* 2. get total number of configured slaves *)
				fbEcGetSlaveCount(bExecute := FALSE);
				fbEcGetSlaveCount(
					sNetId	:= stDriveRef.sNetId,
					bExecute:= TRUE,
					tTimeout:= tTimeout,
				);
				iState		:= iState + 1;
			END_IF
		ELSE
			eFwUpdateState := eFwU_GetSlaveIdentityError;
			bBusy		:= FALSE;
			bError		:= TRUE;
			iErrId		:= fbEcGetSlaveIdentity.nErrId;
			iAdsErrId	:= UDINT_TO_UINT(iErrId);
			iState		:= 0;
		END_IF

		fbEcGetSlaveIdentity(bExecute := FALSE);
	END_IF

2:	(* wait for total number of configured slaves *)
	eFwUpdateState		:= eFwU_CheckSlaveCount;

	fbEcGetSlaveCount();
	IF NOT fbEcGetSlaveCount.bBusy THEN
		IF NOT fbEcGetSlaveCount.bError THEN
			nTotalSlaves:= fbEcGetSlaveCount.nSlaves;
			iState		:= iState + 1;
		ELSE
			eFwUpdateState := eFwU_GetSlaveCountError;
			bBusy		:= FALSE;
			bError		:= TRUE;
			iErrId		:= fbEcGetSlaveCount.nErrId;
			iAdsErrId	:= UDINT_TO_UINT(iErrId);
			iState		:= 0;
		END_IF
		fbEcGetSlaveCount(bExecute := FALSE);
	END_IF

3:	(* 3. get number of next max. 128 configured slave addresses *)
	eFwUpdateState		:= eFwU_CheckFindSlavePos;

	fbAdsRead(
		NETID	:= stDriveRef.sNetId,
		PORT	:= EC_AMSPORT_MASTER,
		IDXGRP	:= EC_ADS_IGRP_CANOPEN_SDO,
		IDXOFFS	:= SHL(nSDO_IDX_SBP_CONFIGUREDSLAVES+nBlockIndex,16) OR 16#00_00_00_00 (*subindex 0*),
		LEN		:= SIZEOF(nSlavesRead),
		DESTADDR:= ADR(nSlavesRead),
		READ	:= TRUE,
		TMOUT	:= tTimeout
	);
	IF NOT fbAdsRead.BUSY THEN
		IF fbAdsRead.ERR THEN
			IF nBlockIndex = 0 THEN
				eFwUpdateState := eFwU_GetSlaveCountError;
				bBusy		:= FALSE;
				bError		:= TRUE;
				iErrId		:= fbAdsRead.ERRID;
				iAdsErrId	:= UDINT_TO_UINT(iErrId);
				iState		:= 0;
			ELSE
				IF fbAdsRead.ERRID = 16#703 THEN
					DelayTimer(IN := FALSE);
					DelayTimer(IN := TRUE, PT := T#0ms);

					(* invalid offset, no next block of 128 slaves available, continue *)
					iState := iState + 2;
				ELSE
					(* report error *)
					bBusy		:= FALSE;
					bError		:= TRUE;
					iErrId		:= fbAdsRead.ERRID;
					iAdsErrId	:= UDINT_TO_UINT(iErrId);
					iState		:= 0;
				END_IF
			END_IF
		ELSE
			nSlaves := nSlaves + nSlavesRead;

			(* 4. get next slave addresses (0xF020 + n) in blocks of 128 *)
			fbCoERead(bExecute := FALSE);
			MEMSET(ADR(nSlaveArr), 0, SIZEOF(nSlaveArr));
			fbCoERead(
				sNetId		:= stDriveRef.sNetId,
				nSlaveAddr	:= EC_AMSPORT_MASTER,
				nSubIndex	:= 0,
				nIndex		:= 16#F020 + nBlockIndex,
				pDstBuf		:= ADR(nSlaveArr),
				cbBufLen	:= SIZEOF(nSlaveArr),
				bExecute	:= TRUE,
				tTimeout	:= tTimeout,
				bCompleteAccess:= TRUE,
			);
			iState	:= iState + 1;

		END_IF;
		fbAdsRead(READ:= FALSE);
	END_IF;

4:	(* wait for slave addresses *)
	fbCoERead();
	IF NOT fbCoERead.bBusy THEN
		IF NOT fbCoERead.bError THEN
			(* find port number *)
			bPositionFound := FALSE;
			FOR I := 0 TO MIN(nSlavesRead, 127) DO
				IF nSlaveArr[I+1] = stDriveRef.nSlaveAddr THEN
					iSlaveIndex := DINT_TO_UINT(I+1);
					iSlaveBlockIndex := nBlockIndex;
					bPositionFound := TRUE;
					EXIT;
				END_IF
			END_FOR

			IF bPositionFound THEN
				IF TestAndSet(bBlockEcatScan) THEN
					iBlockEcatScanCount := iBlockEcatScanCount + 1;

					IF iBlockEcatScanCount = 1 THEN
						bBlockEcatScan := FALSE;
						(* 6. scan revision of AX5000 *)
						(* start scan *)
						nIdxOffs := SHL(nSDO_IDX_SBP_SCANCOMMANDSTART,16) OR 16#00_00_00_01; (* write command *)
						fbAdsWrite(WRITE:= FALSE);
						fbAdsWrite(
							NETID	:= stDriveRef.sNetId,
							PORT	:= EC_AMSPORT_MASTER,
							IDXGRP	:= EC_ADS_IGRP_CANOPEN_SDO,
							IDXOFFS	:= nIdxOffs,
							LEN		:= SIZEOF(nScanCommand),
							SRCADDR	:= ADR(nScanCommand),
							WRITE	:= TRUE,
							TMOUT	:= tTimeout
						);
						iState 		:= iState + 2;
						fbCoERead(bExecute := FALSE);
					ELSE
						IF iBlockEcatScanCount > 0 THEN
							iBlockEcatScanCount := iBlockEcatScanCount - 1;
						END_IF
						bBlockEcatScan := FALSE;
						DelayTimer(IN := FALSE);
						DelayTimer(IN := TRUE, PT := T#100ms);

						(* 5. Delay scan *)
						iState := iState + 1;
						fbCoERead(bExecute := FALSE);
					END_IF
				ELSE
					(* Scanning not blocked, wait *)
					DelayTimer(IN := FALSE);
					DelayTimer(IN := TRUE, PT := T#100ms);

					(* 5. Delay scan *)
					iState := iState + 1;
					fbCoERead(bExecute := FALSE);
				END_IF
			ELSE
				(* read next block of 128 slaves *)
				nBlockIndex := nBlockIndex + 1;
				nSlavesRead := 0;
				iState		:= iState - 1;
				fbCoERead(bExecute := FALSE);
			END_IF
		ELSE
			(* report error *)
			eFwUpdateState := eFwU_GetSlaveAddrError;
			bBusy		:= FALSE;
			bError		:= TRUE;
			iErrId		:= fbCoERead.nErrId;
			iAdsErrId	:= UDINT_TO_UINT(iErrId);
			iState		:= 0;
			fbCoERead(bExecute := FALSE);
		END_IF
	END_IF

5:
	eFwUpdateState		:= eFwU_WaitForScan;

	DelayTimer();
	IF DelayTimer.Q THEN
		DelayTimer(IN := FALSE);

		IF TestAndSet(bBlockEcatScan) THEN
			iBlockEcatScanCount := iBlockEcatScanCount + 1;

			IF iBlockEcatScanCount = 1 THEN
				bBlockEcatScan := FALSE;

				(* 6. scan revision of AX5000 *)
				(* start scan *)
				nIdxOffs := SHL(nSDO_IDX_SBP_SCANCOMMANDSTART,16) OR 16#00_00_00_01; (* write command *)
				fbAdsWrite(WRITE:= FALSE);
				fbAdsWrite(
					NETID	:= stDriveRef.sNetId,
					PORT	:= EC_AMSPORT_MASTER,
					IDXGRP	:= EC_ADS_IGRP_CANOPEN_SDO,
					IDXOFFS	:= nIdxOffs,
					LEN		:= SIZEOF(nScanCommand),
					SRCADDR	:= ADR(nScanCommand),
					WRITE	:= TRUE,
					TMOUT	:= tTimeout
				);
				iState 		:= iState + 1;
			ELSE
				IF iBlockEcatScanCount > 0 THEN
					iBlockEcatScanCount := iBlockEcatScanCount - 1;
				END_IF
				bBlockEcatScan := FALSE;
				DelayTimer(IN := TRUE);
			END_IF
		ELSE
			DelayTimer(IN := TRUE);
		END_IF
	END_IF

6:	(* wait for scan started *)
	eFwUpdateState		:= eFwU_ScanningSlaves;

	fbAdsWrite();
	IF NOT fbAdswrite.BUSY THEN
		IF fbAdsWrite.ERR THEN
			IF TestAndSet(bBlockEcatScan) THEN
				(* Scanning not blocked *)
				IF iBlockEcatScanCount > 0 THEN
					iBlockEcatScanCount := iBlockEcatScanCount - 1;
				END_IF
				bBlockEcatScan := FALSE;
				eFwUpdateState := eFwU_StartScanError;
				bBusy		:= FALSE;
				bError		:= TRUE;
				iErrId		:= fbAdsWrite.ERRID;
				iAdsErrId	:= UDINT_TO_UINT(iErrId);
				iState		:= 0;
			END_IF
		ELSE
			iNoReplyCnt := 0;
			iState := iState + 1; (* 7. wait until command is done *)
		END_IF;
		fbAdsWrite(WRITE:= FALSE);
	END_IF;

7: (* wait until command is done *)
	eFwUpdateState		:= eFwU_ScanningSlaves;

	nIdxOffs := SHL(nSDO_IDX_SBP_SCANCOMMANDSTART,16) OR 16#00_00_00_03; (* read reply *)
	fbAdsRead(
		NETID	:= stDriveRef.sNetId,
		PORT	:= EC_AMSPORT_MASTER,
		IDXGRP	:= EC_ADS_IGRP_CANOPEN_SDO,
		IDXOFFS	:= nIdxOffs,
		LEN		:= SIZEOF(stScanStatus),
		DESTADDR:= ADR(stScanStatus),
		READ	:= TRUE,
		TMOUT	:= tTimeout
	);

	IF NOT fbAdsRead.BUSY THEN
		IF fbAdsRead.ERR THEN
			IF TestAndSet(bBlockEcatScan) THEN
				IF iBlockEcatScanCount > 0 THEN
					iBlockEcatScanCount := iBlockEcatScanCount - 1;
				END_IF
				bBlockEcatScan := FALSE;
				eFwUpdateState := eFwU_ScanStateError;
				bBusy		:= FALSE;
				bError		:= TRUE;
				iErrId		:= fbAdsRead.ERRID;
				iAdsErrId	:= UDINT_TO_UINT(iErrId);
				iState		:= 0;
			END_IF
		ELSE
			IF 	stScanStatus.nScanStatus = eEcScanSlavesCommandState_Completed_NoErrors_NoReply OR
				stScanStatus.nScanStatus = eEcScanSlavesCommandState_Completed_NoErrors_Reply OR
				stScanStatus.nScanStatus = eEcScanSlavesCommandState_Completed_Error_NoReply OR
				stScanStatus.nScanStatus = eEcScanSlavesCommandState_Completed_Error_Reply
			THEN
				IF stScanStatus.nScanStatus = eEcScanSlavesCommandState_Completed_NoErrors_Reply THEN
					eFwUpdateState := eFwU_CheckScannedIdentity;

					(* 8. get scanned data at found position *)
					nIdxOffs := SHL(nSDO_IDX_SBP_SLAVEINFODATASTART+iSlaveBlockIndex*128+iSlaveIndex-1,16) OR nADSIOFFS_ECAT_COE_COMPLETEACCESS;
					fbAdsRead(READ:= FALSE);
					fbAdsRead(
						NETID	:= stDriveRef.sNetId,
						PORT	:= EC_AMSPORT_MASTER,
						IDXGRP	:= EC_ADS_IGRP_CANOPEN_SDO,
						IDXOFFS	:= nIdxOffs,
						LEN		:= SIZEOF(stLocalInfo),
						DESTADDR:= ADR(stLocalInfo),
						READ	:= TRUE,
						TMOUT	:= tTimeout
					);
					iState := iState + 1;
				ELSIF (stScanStatus.nScanStatus = eEcScanSlavesCommandState_Completed_Error_NoReply) AND (iNoReplyCnt < 4) THEN
					iNoReplyCnt := iNoReplyCnt + 1;
					DelayTimer(IN := FALSE);
					iState := 71;
				ELSE
					IF TestAndSet(bBlockEcatScan) THEN
						(* Scanning not blocked *)
						IF iBlockEcatScanCount > 0 THEN
							iBlockEcatScanCount := iBlockEcatScanCount - 1;
						END_IF
						bBlockEcatScan := FALSE;

						eFwUpdateState := eFwU_ScanStateError;
						bBusy		:= FALSE;
						bError		:= TRUE;
						iErrId		:= 16#719;
						iAdsErrId	:= UDINT_TO_UINT(iErrId);
						iState		:= 0;
					END_IF
				END_IF
			ELSE
				iState := iState; (* try it again *)
			END_IF;

		END_IF;
		fbAdsRead(READ:= FALSE);
	END_IF;

71:
	DelayTimer(IN := TRUE, PT:= T#3s);
	IF DelayTimer.Q THEN
		DelayTimer(IN := FALSE);
		iState := 7;
	END_IF


8:	(* wait for scanned data *)
	fbAdsRead();
	IF NOT fbAdsRead.BUSY THEN
		IF TestAndSet(bBlockEcatScan) THEN
			IF iBlockEcatScanCount > 0 THEN
				iBlockEcatScanCount := iBlockEcatScanCount - 1;
			END_IF
			bBlockEcatScan := FALSE;
	
			(*check error and  noOfSlaves > max*)
			IF fbAdsRead.ERR THEN
				eFwUpdateState := eFwU_ScanIdentityError;
				bBusy		:= FALSE;
				bError		:= TRUE;
				iErrId		:= fbAdsRead.ERRID;
				iAdsErrId	:= UDINT_TO_UINT(iErrId);
				iState		:= 0;
			ELSE
				sScannedType:= F_ConvProductCodeToString(stLocalInfo.stSlaveIdentity);
	
				IF (LEFT(sScannedType, 3) <> 'AX5') THEN
					(* scanned slave type <> AX5xxx *)
					eFwUpdateState := eFwU_ScannedTypeInNoAX5xxx;
					bBusy		:= FALSE;
					bError		:= TRUE;
					iErrId		:= 16#70E;
					iAdsErrId	:= UDINT_TO_UINT(iErrId);
					iState		:= 0;
				ELSIF LEFT(sScannedType, 4) <> LEFT(sConfiguredType,4) THEN
					(* mismatch between configured and scanned slave type, e.g. AX52xx <> AX51xx <> AX50xx *)
					IF (LEFT(sConfiguredType, 4) = 'AX51') AND (LEFT(sScannedType, 4) = 'AX52') THEN
						eFwUpdateState := eFwU_ChannelMismatch_1Cfg_2Scanned;
					ELSIF(LEFT(sConfiguredType, 4) = 'AX52') AND (LEFT(sScannedType, 4) = 'AX51') THEN
						eFwUpdateState := eFwU_ChannelMismatch_2Cfg_1Scanned;
					ELSIF (LEFT(sConfiguredType, 4) = 'AX50') AND (LEFT(sScannedType, 4) = 'AX51') THEN
						eFwUpdateState := eFwU_ChannelMismatch_0Cfg_1Scanned;
					ELSIF (LEFT(sConfiguredType, 4) = 'AX50') AND (LEFT(sScannedType, 4) = 'AX52') THEN
						eFwUpdateState := eFwU_ChannelMismatch_0Cfg_2Scanned;
					ELSIF (LEFT(sConfiguredType, 4) = 'AX51') AND (LEFT(sScannedType, 4) = 'AX50') THEN
						eFwUpdateState := eFwU_ChannelMismatch_1Cfg_0Scanned;
					ELSIF (LEFT(sConfiguredType, 4) = 'AX52') AND (LEFT(sScannedType, 4) = 'AX50') THEN
						eFwUpdateState := eFwU_ChannelMismatch_2Cfg_0Scanned;
					ELSE
						eFwUpdateState := eFwU_ChannelMismatch;
					END_IF

					bBusy		:= FALSE;
					bError		:= TRUE;
					iErrId		:= 16#70E;
					iAdsErrId	:= UDINT_TO_UINT(iErrId);
					iState		:= 0;
				ELSIF (MID(sConfiguredType, 2, 5) <> MID(sScannedType, 2, 5)) AND
					(	((LEFT(sConfiguredType, 4) = 'AX51') AND (LEFT(sScannedType, 4) = 'AX51')) OR
						((LEFT(sConfiguredType, 4) = 'AX52') AND (LEFT(sScannedType, 4) = 'AX52'))	) THEN

					eFwUpdateState := eFwU_CurrentMismatch;
	
					bBusy		:= FALSE;
					bError		:= TRUE;
					iErrId		:= 16#70E;
					iAdsErrId	:= UDINT_TO_UINT(iErrId);
					iState		:= 0;
				ELSE
					(* create firmware file name *)
					sScannedFirmwareFile 	:= '';
					sScannedFirmwareFileDUC := '';
					IF (LEFT(sScannedType, 4) = 'AX50') THEN
						sScannedFirmwareFile := LEFT(sScannedType, 6);								(* --> "AX5021"               *)
						sScannedFirmwareFile := CONCAT(sScannedFirmwareFile, '_xxxx_');				(* --> "AX5021_xxxx_"         *)
					ELSIF (LEFT(sScannedType, 4) = 'AX51') OR (LEFT(sScannedType, 4) = 'AX52') THEN
						sScannedFirmwareFile := 'AX5yxx_xxxx_';									(* --> "AX5yxx_xxxx_"         *)
					END_IF

					sScannedFirmwareFile 	:= CONCAT(sScannedFirmwareFile, RIGHT(sScannedType,4));	(* --> "AX5021_xxxx_0002"                 or "AX5yxx_xxxx_0010"   *)
					sScannedFirmwareFile 	:= CONCAT(sScannedFirmwareFile, '_');					(* --> "AX5021_xxxx_0002_"                or "AX5yxx_xxxx_0010_"  *)
					sScannedFirmwareFileDUC := sScannedFirmwareFile;
					sScannedFirmwareFile 	:= F_ToUCase(sScannedFirmwareFile);
					sScannedFirmwareFileDUC	:= F_ToUCase(sScannedFirmwareFileDUC);
					
					iState 	:= iState + 1;
					eFwUpdateState := eFwU_CheckScannedFirmware;

					(* 9. check slave state *)
					fbEcGetSlaveState(bExecute := FALSE);
					fbEcGetSlaveState(
						sNetId		:= stDriveRef.sNetId,
						nSlaveAddr	:= stDriveRef.nSlaveAddr,
						bExecute	:= TRUE,
						tTimeout	:= tTimeout,
					);
				END_IF
			END_IF;
			fbAdsRead(READ:= FALSE);
		END_IF
	END_IF;

9:	(* wait for slave state *)
	fbEcGetSlaveState();
	IF NOT fbEcGetSlaveState.bBusy THEN
		IF fbEcGetSlaveState.bError THEN
			eFwUpdateState := eFwU_GetSlaveStateError;
			bBusy		:= FALSE;
			bError		:= TRUE;
			iErrId		:= fbEcGetSlaveState.nErrId;
			iAdsErrId	:= UDINT_TO_UINT(iErrId);
			iState		:= 0;
		ELSE
			iSlaveState := fbEcGetSlaveState.state.deviceState;

			IF ((iSlaveState AND EC_DEVICE_STATE_INVALID_VPRS) <> EC_DEVICE_STATE_INVALID_VPRS) AND
				(((iSlaveState AND 16#0F) = EC_DEVICE_STATE_PREOP) OR ((iSlaveState AND 16#0F) >= EC_DEVICE_STATE_SAFEOP)) THEN

				(* 10. get firmware version *)
				fbGetSwSoE(bExecute:= FALSE);
				fbGetSwSoE(
					stDriveRef	:= stDriveRef,
					nIdn		:= S_0_IDN + 30,
					nElement	:= EC_SOE_ELEMENT_VALUE,
					pDstBuf		:= ADR(stSoEValue),
					cbBufLen	:= SIZEOF(stSoEValue),
					bExecute	:= TRUE,
					tTimeout	:= tTimeout,
				);
				iState 	:= iState + 1;
			ELSE
				(* no SoE communication possible due to VPRS error *)
				sScannedFirmwareFile 	:= CONCAT(sScannedFirmwareFile, 'v?_??_b00??.efw');						(* --> "AX5021_xxxx_0002_v?_??_b00??.efw" 					or "AX5yxx_xxxx_0010_v?_??_b00??.efw"  *)
				sScannedFirmwareFileDUC := CONCAT(sScannedFirmwareFileDUC, 'v?_??_b00??_dual_use_conform.efw');	(* --> "AX5021_xxxx_0002_v?_??_b00??_dual_use_conform.efw" 	or "AX5yxx_xxxx_0010_v?_??_b00??_dual_use_conform.efw"  *)
				sScannedFirmwareFile 	:= F_ToUCase(sScannedFirmwareFile);
				sScannedFirmwareFileDUC	:= F_ToUCase(sScannedFirmwareFileDUC);
				iState 	:= iState + 2;

				(* 11. search firmware file(s) *)
				bExecFind					:= TRUE;
				iFilesFound 				:= 0;
				sSelectedFirmwareFile		:= '';
				sFoundFirmwareFile			:= '';
				fbFindFiles(bExecute := FALSE);
				fbFindFiles.sNetId			:= sNetIdIPC;
				fbFindFiles.eCmd 			:= eEnumCmd_First;
				fbFindFiles.sPathName 		:= CONCAT(sFirmwarePath, '\');
				sCompatibleFirmwareFile 	:= '';

				bExecFindDUC				:= TRUE;
				iFilesFoundDUC 				:= 0;
				sSelectedFirmwareFileDUC	:= '';
				sFoundFirmwareFileDUC		:= '';
				fbFindFilesDUC(bExecute := FALSE);
				fbFindFilesDUC.sNetId		:= sNetIdIPC;
				fbFindFilesDUC.eCmd 		:= eEnumCmd_First;
				fbFindFilesDUC.sPathName 	:= CONCAT(sFirmwarePath, '\');
				sCompatibleFirmwareFileDUC	:= '';

				bCompatibleMode 			:= FALSE;
				bIncompatibleType 			:= FALSE;

				(* check for same or compatible version *)
				IF (RIGHT(sScannedType,4) >= '0200' AND RIGHT(sConfiguredType,4) < '0200') THEN
					(* scanned revision HW >= 2 and configured revision HW =  1 *)
					(* sCompatibleFirmwareFile 	:=            'AX5yxx_xxxx_0200'       +          '_v?_??_b00??.efw' *)
					sCompatibleFirmwareFile 	:= CONCAT(LEFT(sScannedFirmwareFile, 16), 	 RIGHT(sConfiguredFirmwareFile, 16));
					fbFindFiles.sPathName 		:= CONCAT(fbFindFiles.sPathName, sCompatibleFirmwareFile);
					(* sCompatibleFirmwareFileDUC:=           'AX5yxx_xxxx_0200'       +          '_v?_??_b00??_dual_use_conform.efw' *)
					sCompatibleFirmwareFileDUC 	:= CONCAT(LEFT(sScannedFirmwareFileDUC, 16), RIGHT(sConfiguredFirmwareFileDUC, 33));
					fbFindFilesDUC.sPathName	:= CONCAT(fbFindFilesDUC.sPathName, sCompatibleFirmwareFileDUC);
					sCompatibleFirmwareFile 	:= F_ToUCase(sCompatibleFirmwareFile);
					sCompatibleFirmwareFileDUC	:= F_ToUCase(sCompatibleFirmwareFileDUC);
					bCompatibleMode 			:= TRUE;

				ELSIF RIGHT(sScannedType,4) < '0200' AND RIGHT(sConfiguredType,4) < '0200' OR
					(RIGHT(sScannedType,4) >= '0200' AND RIGHT(sConfiguredType,4) >= '0200') THEN
					(* scanned revision HW =  1 and configured revision HW =  1 or scanned revision HW =  2 and configured revision HW =  2 *)
					fbFindFiles.sPathName 		:= CONCAT(fbFindFiles.sPathName, sConfiguredFirmwareFile);
					fbFindFilesDUC.sPathName 	:= CONCAT(fbFindFilesDUC.sPathName, sConfiguredFirmwareFileDUC);
				ELSE (* RIGHT(sScannedType,4) < '0200' AND RIGHT(sConfiguredType,4) >= '0200' *)
					(* scanned revision HW =  1 and configured revision HW >= 2 *)
					(* sCompatibleFirmwareFile 	:=         	  'AX5yxx_xxxx_0010'       +   	      '_v?_??_b00??.efw' *)
					sCompatibleFirmwareFile 	:= CONCAT(LEFT(sScannedFirmwareFile, 16), 	 RIGHT(sConfiguredFirmwareFile, 16));
					(* sCompatibleFirmwareFileDUC:=           'AX5yxx_xxxx_0010'       +          '_v?_??_b00??_dual_use_conform.efw' *)
					sCompatibleFirmwareFileDUC 	:= CONCAT(LEFT(sScannedFirmwareFileDUC, 16), RIGHT(sConfiguredFirmwareFileDUC, 33));
					sCompatibleFirmwareFile 	:= F_ToUCase(sCompatibleFirmwareFile);
					sCompatibleFirmwareFileDUC	:= F_ToUCase(sCompatibleFirmwareFileDUC);
					bIncompatibleType 			:= TRUE;
				END_IF

				IF bIncompatibleType THEN
					(* incompatible HW 1 scanned but HW 2 configured, no download possible *)
					eFwUpdateState := eFwU_TypeIncompatibleCfgToScanned;
					bBusy	:= FALSE;
					iState	:= 0;
				END_IF
			END_IF
		END_IF
		fbEcGetSlaveState(bExecute := FALSE);
	END_IF

10:	(* wait for scanned firmware version of AX5000 *)
	fbGetSwSoE();
	IF NOT fbGetSwSoE.bBusy THEN
		IF fbGetSwSoE.bError THEN
			eFwUpdateState := eFwU_ScanFirmwareError;
			bBusy		:= FALSE;
			bError		:= TRUE;
			iAdsErrId	:= fbGetSwSoE.iAdsErrId;
			iSercosErrId:= fbGetSwSoE.iSercosErrId;
			iState		:= 0;
		ELSE
			sScannedFirmwareVersion := stSoEValue.strData;

			(* parse firmware string, e.g. "Firmware: v1.05 (Build 0009) / Bootloader: v1.02 (Build 0001)" *)
			iStrPosV 		 := FIND(sScannedFirmwareVersion, 'v');
			iStrPosBuild 	 := FIND(sScannedFirmwareVersion, ' (Build ');
			sTemp 			 := MID(sScannedFirmwareVersion, iStrPosBuild-iStrPosV, iStrPosV); (* --> "v1.05" *)
			iStrPosDot 		 := FIND(sTemp, '.');

			sScannedVBString := LEFT(sTemp, iStrPosDot-1); 		(* --> "v1" *)
			sScannedVBString := CONCAT(sScannedVBString, '_'); 	(* --> "v1_" *)
			sScannedVBString := CONCAT(sScannedVBString, RIGHT(sTemp, LEN(sTemp)-iStrPosDot)); 							(* --> "v1_05" *)
			sScannedVBString := CONCAT(sScannedVBString, '_b');															(* --> "v1_05_b" *)
			sScannedVBString := CONCAT(sScannedVBString, MID(sScannedFirmwareVersion, 4, iStrPosBuild+LEN(' (Build ')));(* --> "v1_05_b0009" *)

			sScannedFirmwareFile 		:= CONCAT(sScannedFirmwareFile, sScannedVBString);			   (* --> "AX5021_xxxx_0002_v1_05_b0009" or 						"AX5yxx_xxxx_0010_v1_05_b0009" *)
			sScannedFirmwareFileDUC 	:= CONCAT(sScannedFirmwareFileDUC, sScannedVBString);		   (* --> "AX5021_xxxx_0002_v1_05_b0009" or 						"AX5yxx_xxxx_0010_v1_05_b0009" *)
			sScannedFirmwareFile 		:= CONCAT(sScannedFirmwareFile, '.efw');					   (* --> "AX5021_xxxx_0002_v1_05_b0009.efw" OR 					"AX5yxx_xxxx_0010_v1_05_b0009.efw" *)
			sScannedFirmwareFileDUC 	:= CONCAT(sScannedFirmwareFileDUC, '_dual_use_conform.efw');   (* --> "AX5021_xxxx_0002_v1_05_b0009_dual_use_conform.efw" or 	"AX5yxx_xxxx_0010_v1_05_b0009_dual_use_conform.efw" *)
			sScannedFirmwareFile 		:= F_ToUCase(sScannedFirmwareFile);
			sScannedFirmwareFileDUC		:= F_ToUCase(sScannedFirmwareFileDUC);
			sCompatibleFirmwareFile 	:= '';
			sCompatibleFirmwareFileDUC 	:= '';
			bCompatibleMode 			:= FALSE;
			bIncompatibleType 			:= FALSE;

			(* check for same or compatible version *)
			IF (RIGHT(sScannedType,4) >= '0200' AND RIGHT(sConfiguredType,4) < '0200') THEN
				(* scanned revision HW >= 2 and configured revision HW =  1 *)
				(* sCompatibleFirmwareFile 	:=            'AX5yxx_xxxx_0200'       +         '_v2_03_b0026.efw' *)
				sCompatibleFirmwareFile 	:= CONCAT(LEFT(sScannedFirmwareFile, 16), 	RIGHT(sConfiguredFirmwareFile, 16));
				(* sCompatibleFirmwareFileDUC:=           'AX5yxx_xxxx_0200'       +         '_v2_03_b0026_dual_use_conform.efw' *)
				sCompatibleFirmwareFileDUC 	:= CONCAT(LEFT(sScannedFirmwareFileDUC, 16),RIGHT(sConfiguredFirmwareFileDUC, 33));
				sCompatibleFirmwareFile 	:= F_ToUCase(sCompatibleFirmwareFile);
				sCompatibleFirmwareFileDUC	:= F_ToUCase(sCompatibleFirmwareFileDUC);

				bCompatibleMode 		:= TRUE;
			ELSIF RIGHT(sScannedType,4) < '0200' AND RIGHT(sConfiguredType,4) < '0200' OR
				(RIGHT(sScannedType,4) >= '0200' AND RIGHT(sConfiguredType,4) >= '0200') THEN
				(* scanned revision HW =  1 and configured revision HW =  1 or scanned revision HW =  2 and configured revision HW =  2 *)
				;
			ELSE (* RIGHT(sScannedType,4) < '0200' AND RIGHT(sConfiguredType,4) >= '0200' *)
				(* scanned revision HW =  1 and configured revision HW >= 2 *)
				(* sCompatibleFirmwareFile  :=            'AX5yxx_xxxx_0010'       +         '_v2_03_b0026.efw' *)
				sCompatibleFirmwareFile 	:= CONCAT(LEFT(sScannedFirmwareFile, 16), 	RIGHT(sConfiguredFirmwareFile, 16));
				(* sCompatibleFirmwareFileDUC:=           'AX5yxx_xxxx_0010'       +         '_v2_03_b0026_dual_use_conform.efw' *)
				sCompatibleFirmwareFileDUC 	:= CONCAT(LEFT(sScannedFirmwareFileDUC, 16),RIGHT(sConfiguredFirmwareFileDUC, 33));
				sCompatibleFirmwareFile 	:= F_ToUCase(sCompatibleFirmwareFile);
				sCompatibleFirmwareFileDUC	:= F_ToUCase(sCompatibleFirmwareFileDUC);

				bIncompatibleType 		:= TRUE;
			END_IF

			(* verify firmware version *)
			IF (sScannedFirmwareFile = sConfiguredFirmwareFile) AND (sScannedFirmwareFileDUC = sConfiguredFirmwareFileDUC) THEN
				(* no download required *)
				eFwUpdateState := eFwU_NoFwUpdateRequired;
				bBusy	:= FALSE;
				iState	:= 0;

			ELSIF bIncompatibleType THEN
				(* incompatible HW 1 scanned but HW 2 configured, no download possible *)
				eFwUpdateState := eFwU_TypeIncompatibleCfgToScanned;
				bBusy	:= FALSE;
				iState	:= 0;
			
			ELSIF bCompatibleMode AND (sScannedFirmwareFile = sCompatibleFirmwareFile) AND (sScannedFirmwareFileDUC = sConfiguredFirmwareFileDUC) THEN
				(* compatibility mode, no download required *)
				eFwUpdateState := eFwU_NoFwUpdateRequired;
				bBusy	:= FALSE;
				iState	:= 0;
				
			ELSE
				(* 13. search firmware file(s) *)
				bExecFind				:= TRUE;
				iFilesFound 			:= 0;
				sSelectedFirmwareFile	:= '';
				sFoundFirmwareFile		:= '';
				fbFindFiles(bExecute := FALSE);
				fbFindFiles.sNetId		:= sNetIdIPC;
				fbFindFiles.eCmd 		:= eEnumCmd_First;
				fbFindFiles.sPathName 	:= CONCAT(sFirmwarePath, '\');

				bExecFindDUC			:= TRUE;
				iFilesFoundDUC 			:= 0;
				sSelectedFirmwareFileDUC:= '';
				sFoundFirmwareFileDUC	:= '';
				fbFindFilesDUC(bExecute := FALSE);
				fbFindFilesDUC.sNetId	:= sNetIdIPC;
				fbFindFilesDUC.eCmd 	:= eEnumCmd_First;
				fbFindFilesDUC.sPathName:= CONCAT(sFirmwarePath, '\');

				IF bCompatibleMode THEN
					(* find compatible firmware file *)
					fbFindFiles.sPathName := CONCAT(fbFindFiles.sPathName, sCompatibleFirmwareFile);
					fbFindFilesDUC.sPathName:= CONCAT(fbFindFilesDUC.sPathName, sCompatibleFirmwareFileDUC);
				ELSE
					(* find configured firmware file *)
					fbFindFiles.sPathName := CONCAT(fbFindFiles.sPathName, sConfiguredFirmwareFile);
					fbFindFilesDUC.sPathName:= CONCAT(fbFindFilesDUC.sPathName, sConfiguredFirmwareFileDUC);
				END_IF
				iState 	:= iState + 1;
			END_IF
		END_IF

		fbGetSwSoE(bExecute:= FALSE);
	END_IF

11:	(* search firmware file(s) *)
	eFwUpdateState := eFwU_FindFirmwareFile;

	fbFindFiles(bExecute := FALSE);
	fbFindFiles(
		bExecute	:= bExecFind,
		tTimeout	:= tTimeout,
	);

	fbFindFilesDUC(bExecute := FALSE);
	fbFindFilesDUC(
		bExecute	:= bExecFindDUC,
		tTimeout	:= tTimeout,
	);

	iState 	:= iState + 1;

12: (* wait for search firmware file(s) *)
	fbFindFiles( bExecute := FALSE, bEOE=>bNoMoreFiles );
	fbFindFilesDUC( bExecute := FALSE, bEOE=>bNoMoreFilesDUC );

	IF NOT fbFindFiles.bBusy AND NOT fbFindFilesDUC.bBusy THEN
		IF bNoMoreFiles THEN
			bExecFind 	:= FALSE;
		END_IF
		IF bNoMoreFilesDUC  THEN
			bExecFindDUC:= FALSE;
		END_IF

		IF (NOT bExecFind AND NOT bExecFindDUC) THEN
			(* nothing more available to be found *)

			IF fbFindFiles.bError AND (sFoundFirmwareFileDUC = '') THEN
				eFwUpdateState := eFwU_FindFileError;
				IF bCompatibleMode THEN
					sSelectedFirmwareFile := sCompatibleFirmwareFile;
				ELSE
					sSelectedFirmwareFile := sConfiguredFirmwareFile;
				END_IF
				bBusy		:= FALSE;
				bError		:= TRUE;
				iErrId		:= fbFindFiles.nErrID;
				iAdsErrId	:= UDINT_TO_UINT(iErrId);
				iState		:= 0;
			ELSIF fbFindFilesDUC.bError AND (sFoundFirmwareFile = '') THEN
				eFwUpdateState := eFwU_FindFileError;
				IF bCompatibleMode THEN
					sSelectedFirmwareFile := sCompatibleFirmwareFileDUC;
				ELSE
					sSelectedFirmwareFile := sConfiguredFirmwareFileDUC;
				END_IF
				bBusy		:= FALSE;
				bError		:= TRUE;
				iErrId		:= fbFindFilesDUC.nErrID;
				iAdsErrId	:= UDINT_TO_UINT(iErrId);
				iState		:= 0;
			END_IF

			IF NOT bError THEN
				IF (sFoundFirmwareFile = '' AND sFoundFirmwareFileDUC = '') THEN
					(* firmware update file(s) not found *)
					eFwUpdateState := eFwU_FindFileError;
					IF bCompatibleMode THEN
						sSelectedFirmwareFile 	:= sCompatibleFirmwareFile;
						sSelectedFirmwareFileDUC:= sCompatibleFirmwareFileDUC;
					ELSE
						sSelectedFirmwareFile 	:= sConfiguredFirmwareFile;
						sSelectedFirmwareFileDUC:= sConfiguredFirmwareFileDUC;
					END_IF
					bBusy		:= FALSE;
					bError		:= TRUE;
					iErrId		:= 16#70C;
					iAdsErrId	:= UDINT_TO_UINT(iErrId);
					iState		:= 0;
				ELSE
					IF (sScannedFirmwareFile = sSelectedFirmwareFile) AND (sSelectedFirmwareFile <> '') AND
						(sScannedFirmwareFileDUC = sSelectedFirmwareFileDUC) AND (sSelectedFirmwareFileDUC <> '') AND
						(LEFT(sSelectedFirmwareFile, 28) = LEFT(sScannedFirmwareFileDUC, 28)) THEN

						(* no download required *)
						eFwUpdateState := eFwU_NoFwUpdateRequired;
						bBusy	:= FALSE;
						iState	:= 0;

					ELSIF (sScannedFirmwareFile = sSelectedFirmwareFile) AND (sSelectedFirmwareFile <> '') AND (sSelectedFirmwareFileDUC = '') THEN
						(* no download required *)
						eFwUpdateState := eFwU_NoFwUpdateRequired;
						bBusy	:= FALSE;
						iState	:= 0;
					ELSIF (sScannedFirmwareFileDUC = sSelectedFirmwareFileDUC) AND (sSelectedFirmwareFileDUC <> '') AND (sSelectedFirmwareFile = '') THEN
						(* no download required *)
						sSelectedFirmwareFile := sSelectedFirmwareFileDUC;
						eFwUpdateState := eFwU_NoFwUpdateRequired;
						bBusy	:= FALSE;
						iState	:= 0;

					ELSIF (sScannedFirmwareFile = sSelectedFirmwareFile) AND (LEFT(sSelectedFirmwareFile, 28) >= LEFT(sSelectedFirmwareFileDUC, 28)) AND bUseLatestBuild THEN
						(* no download required *)
						eFwUpdateState := eFwU_NoFwUpdateRequired;
						bBusy	:= FALSE;
						iState	:= 0;
					ELSIF (sScannedFirmwareFileDUC = sSelectedFirmwareFileDUC) AND (LEFT(sSelectedFirmwareFileDUC, 28) >= LEFT(sSelectedFirmwareFile, 28)) AND bUseLatestBuild THEN
						(* no download required *)
						sSelectedFirmwareFile := sSelectedFirmwareFileDUC;
						eFwUpdateState := eFwU_NoFwUpdateRequired;
						bBusy	:= FALSE;
						iState	:= 0;

					ELSE
						(* 13. check for update *)
						IF sSelectedFirmwareFile = '' THEN
							sSelectedFirmwareFile := sSelectedFirmwareFileDUC;
						ELSIF sSelectedFirmwareFileDUC = '' THEN
							sSelectedFirmwareFileDUC := sSelectedFirmwareFile;
						ELSIF (LEFT(sSelectedFirmwareFile, 28) < LEFT(sSelectedFirmwareFileDUC, 28)) AND bUseLatestBuild THEN
							sSelectedFirmwareFile := sFoundFirmwareFileDUC;
						END_IF

						eFwUpdateState:= eFwU_WaitForUpdate;
						iState := iState + 1;
					END_IF
				END_IF
			END_IF
		ELSE
			(* continue search *)
			IF bExecFind THEN
				(* evaluate data *)
				sFoundFirmwareFile	:= fbFindFiles.stFindFile.sFileName;
				sFoundFirmwareFile 	:= F_ToUCase(sFoundFirmwareFile);
				IF sSelectedFirmwareFile = '' THEN
					sSelectedFirmwareFile := sFoundFirmwareFile;
				ELSIF (sSelectedFirmwareFile < sFoundFirmwareFile) AND bUseLatestBuild THEN
					sSelectedFirmwareFile := sFoundFirmwareFile;
				END_IF

				iFilesFound	:= iFilesFound + 1;
				fbFindFiles.eCmd := eEnumCmd_Next;
			END_IF

			IF bExecFindDUC THEN
				(* evaluate data *)
				sFoundFirmwareFileDUC:= fbFindFilesDUC.stFindFile.sFileName;
				sFoundFirmwareFileDUC:= F_ToUCase(sFoundFirmwareFileDUC);
				IF sSelectedFirmwareFileDUC = '' THEN
					sSelectedFirmwareFileDUC := sFoundFirmwareFileDUC;
				ELSIF (sSelectedFirmwareFileDUC < sFoundFirmwareFileDUC) AND bUseLatestBuild THEN
					sSelectedFirmwareFileDUC := sFoundFirmwareFileDUC;
				END_IF

				iFilesFoundDUC	:= iFilesFoundDUC + 1;
				fbFindFilesDUC.eCmd := eEnumCmd_Next;
			END_IF
			iState := iState - 1;
		END_IF
		fbFindFiles( bExecute := FALSE, bEOE=>bNoMoreFiles );
		fbFindFilesDUC( bExecute := FALSE, bEOE=>bNoMoreFilesDUC );
	END_IF

13:	(* check for update *)
	eFwUpdateState:= eFwU_WaitForUpdate;

	IF TestAndSet(bBlockDrivesFwUpdate) THEN
		(* Firmwareupdate not blocked *)
		iNextUpdateIdx	:= -1;
		iCurUpdateIdx	:= -1;

		FOR I := 0 TO iMaxNumOfDrivesUpdate DO
			IF iArrDrivesUpdatePorts[I] = stDriveRef.nSlaveAddr THEN
				eFwUpdateState		:= eFwU_UpdateViaOtherChannelActive;
				bUpdateViaOtherChn 	:= TRUE;
				iCurUpdateIdx		:= DINT_TO_INT(I);
				EXIT;
			ELSIF (iArrDrivesUpdatePorts[I] = 0) AND (iNextUpdateIdx = -1) THEN
				iNextUpdateIdx	:= DINT_TO_INT(I);
			END_IF
		END_FOR

		IF iCurUpdateIdx = -1 THEN
			iCurUpdateIdx := 0;
		END_IF
		IF iNextUpdateIdx = -1 THEN
			iNextUpdateIdx := 0;
		END_IF

		IF bUpdateViaOtherChn THEN
			bBlockDrivesFwUpdate := FALSE;

			(* update via other channel *)
			iState := 19;
		ELSE
			iArrDrivesUpdatePorts[iNextUpdateIdx] := stDriveRef.nSlaveAddr;
			bBlockDrivesFwUpdate := FALSE;

			(* update *)
			iState := iState + 1;
			DelayTimer(IN := FALSE);
			DelayTimer(IN := TRUE, PT := T#10s);
		END_IF
	END_IF

14:
	DelayTimer();
	IF DelayTimer.Q THEN
		IF TestAndSet(bBlockEcatScan) THEN
			iBlockEcatScanCount := iBlockEcatScanCount + 1;
			bBlockEcatScan := FALSE;

			(* 15. Update Firmware *)
			eFwUpdateState := eFwU_StartFwUpdate;
		
			fbEcFoeLoad(bExecute := FALSE);
			fbEcFoeLoad.sPathName 	:= CONCAT(sFirmwarePath, '\');
			fbEcFoeLoad.sPathName 	:= CONCAT(fbEcFoeLoad.sPathName, sSelectedFirmwareFile);
			fbEcFoeLoad(
				sNetId		:= stDriveRef.sNetId,
				nSlaveAddr	:= stDriveRef.nSlaveAddr,
				bExecute	:= TRUE
			);
			iState := iState + 1;
		END_IF
	END_IF

15:	(* wait for Firmware Update done *)
	eFwUpdateState := eFwU_FwUpdateInProgress;

	fbEcFoeLoad();
	iLoadProgress := UDINT_TO_INT(fbEcFoeLoad.nProgress);

	IF NOT fbEcFoeLoad.bBusy THEN
		IF fbEcFoeLoad.bError THEN
			iState 		:= iState + 1;
			iErrId		:= fbEcFoeLoad.nErrId;
			iAdsErrId	:= UDINT_TO_UINT(iErrId);

			(* get error number from info string *)
			iFindStrPos := FIND(fbEcFoeLoad.sInfo, 'Error Code: '); (* "Download failed! (AX5000 Error Code: F077)" *)
			IF (iFindStrPos <> 0) AND LEN(fbEcFoeLoad.sInfo) >= iFindStrPos + 16 THEN
				sFoEInfo := F_ToUCase(MID(fbEcFoeLoad.sInfo, 4, iFindStrPos + 12));(* "F077" *)
				MEMCPY(ADR(iByteArr4), ADR(sFoEInfo), SIZEOF(iByteArr4));

				FOR I := 0 TO 3 DO
					IF iByteArr4[I] >= 16#30 AND iByteArr4[I] <= 16#39 THEN
						(* number *)
						iByteArr4[I] := iByteArr4[I] - 16#30;
					ELSIF iByteArr4[I] >= 65 AND iByteArr4[I] <= 70 THEN
						(* letter A..F *)
						iByteArr4[I] := iByteArr4[I] - 55;
					ELSE
						MEMSET(ADR(iByteArr4), 0, SIZEOF(iByteArr4));
						EXIT;
					END_IF
				END_FOR

				iDiagNumber := iByteArr4[3] + iByteArr4[2] * 16 + iByteArr4[1] * 256 + iByteArr4[0] * 4096;
			END_IF

			(* 16. request INIT slave state *)
			fbEcReqSlaveState(bExecute := FALSE);
			fbEcReqSlaveState(
				sNetId		:= stDriveRef.sNetId,
				nSlaveAddr	:= stDriveRef.nSlaveAddr,
				bExecute	:= TRUE,
				tTimeout	:= tTimeout,
				state		:= EC_DEVICE_STATE_INIT,
			);
		ELSE
			iState := iState + 2;

			(* 18. check slave state *)
			fbEcGetSlaveState(bExecute := FALSE);
			fbEcGetSlaveState(
				sNetId		:= stDriveRef.sNetId,
				nSlaveAddr	:= stDriveRef.nSlaveAddr,
				bExecute	:= TRUE,
				tTimeout	:= tTimeout,
			);
		END_IF

		fbEcFoeLoad(bExecute := FALSE);
	END_IF

16:	(* request INIT slave state *)
	eFwUpdateState := eFwU_WaitForSlaveState;

	fbEcReqSlaveState();
	IF NOT fbEcReqSlaveState.bBusy THEN
		IF TestAndSet(bBlockEcatScan) THEN
			IF iBlockEcatScanCount > 0 THEN
				iBlockEcatScanCount := iBlockEcatScanCount - 1;
			END_IF
			bBlockEcatScan := FALSE;
			eFwUpdateState := eFwU_FwUpdateError;
			bError		:= TRUE;
			iState		:= 25;
	
			fbEcReqSlaveState(bExecute := FALSE);
		END_IF
	END_IF

17:	(* wait for boot *)
	eFwUpdateState := eFwU_WaitForSlaveState;

	fbEcGetSlaveState();
	IF NOT fbEcGetSlaveState.bBusy THEN
		IF fbEcGetSlaveState.bError THEN
			IF TestAndSet(bBlockEcatScan) THEN
				IF iBlockEcatScanCount > 0 THEN
					iBlockEcatScanCount := iBlockEcatScanCount - 1;
				END_IF
				bBlockEcatScan := FALSE;
				eFwUpdateState := eFwU_GetSlaveStateError;
				bError		:= TRUE;
				iErrId		:= fbEcGetSlaveState.nErrId;
				iAdsErrId	:= UDINT_TO_UINT(iErrId);
				iState		:= 25;
			END_IF
		ELSE
			iSlaveState := fbEcGetSlaveState.state.deviceState;

			IF (iSlaveState = iReqEcState) THEN
				IF TestAndSet(bBlockEcatScan) THEN
					IF iBlockEcatScanCount > 0 THEN
						iBlockEcatScanCount := iBlockEcatScanCount - 1;
					END_IF
					bBlockEcatScan := FALSE;
					DelayTimer(IN := FALSE);
					DelayTimer(IN := TRUE, PT := T#0s);
					iState	:= 21;
				END_IF
			ELSE
				iState := iState + 1;

				(* 18. Request slave state *)
				fbEcReqSlaveState(bExecute := FALSE);
				fbEcReqSlaveState(
					sNetId		:= stDriveRef.sNetId,
					nSlaveAddr	:= stDriveRef.nSlaveAddr,
					bExecute	:= TRUE,
					tTimeout	:= tTimeout,
					state		:= iReqEcState,
				);
			END_IF
		END_IF
	END_IF

18:	(* wait for slave state *)
	eFwUpdateState := eFwU_WaitForSlaveState;

	fbEcReqSlaveState();
	IF NOT fbEcReqSlaveState.bBusy THEN
		IF TestAndSet(bBlockEcatScan) THEN
			IF iBlockEcatScanCount > 0 THEN
				iBlockEcatScanCount := iBlockEcatScanCount - 1;
			END_IF
			bBlockEcatScan := FALSE;
			IF fbEcReqSlaveState.bError THEN
				eFwUpdateState := eFwU_ReqSlaveStateError;
				bError		:= TRUE;
				iErrId		:= fbEcReqSlaveState.nErrId;
				iAdsErrId	:= UDINT_TO_UINT(iErrId);
				iState		:= 25;
			ELSE
				DelayTimer(IN := FALSE);
				DelayTimer(IN := TRUE, PT := T#0s);
				iState := 21;
			END_IF
			fbEcReqSlaveState(bExecute := FALSE);
		END_IF
	END_IF

19:
	(* 13 --> 19 update via other channel *)
	IF TestAndSet(bBlockDrivesFwUpdate) THEN
		(* Firmwareupdate not blocked *)
		IF iArrDrivesUpdatePorts[iCurUpdateIdx] = stDriveRef.nSlaveAddr THEN
			DelayTimer(IN := FALSE);
			DelayTimer(IN := TRUE, PT := T#100ms);
			iState := iState + 1;
		ELSE
			DelayTimer(IN := FALSE);
			DelayTimer(IN := TRUE, PT := T#100ms);
			iState := iState + 2;
		END_IF
		bBlockDrivesFwUpdate := FALSE;
	END_IF

20:
	DelayTimer();
	IF DelayTimer.Q THEN
		DelayTimer(IN := FALSE);
		iState := iState - 1;
	END_IF

21:
	(* 17, 18, 19 --> 21 rescan *)
	eFwUpdateState := eFwU_WaitForScan;

	DelayTimer();
	IF DelayTimer.Q THEN
		DelayTimer(IN := FALSE);

		IF TestAndSet(bBlockEcatScan) THEN
			iBlockEcatScanCount := iBlockEcatScanCount + 1;

			IF iBlockEcatScanCount = 1 THEN
				bBlockEcatScan := FALSE;

				(* 22. scan revision of AX5000 *)
				(* start scan *)
				nIdxOffs := SHL(nSDO_IDX_SBP_SCANCOMMANDSTART,16) OR 16#00_00_00_01; (* write command *)
				fbAdsWrite(WRITE:= FALSE);
				fbAdsWrite(
					NETID	:= stDriveRef.sNetId,
					PORT	:= EC_AMSPORT_MASTER,
					IDXGRP	:= EC_ADS_IGRP_CANOPEN_SDO,
					IDXOFFS	:= nIdxOffs,
					LEN		:= SIZEOF(nScanCommand),
					SRCADDR	:= ADR(nScanCommand),
					WRITE	:= TRUE,
					TMOUT	:= tTimeout
				);
				iState 		:= iState + 1;
			ELSE
				IF iBlockEcatScanCount > 0 THEN
					iBlockEcatScanCount := iBlockEcatScanCount - 1;
				END_IF
				bBlockEcatScan := FALSE;
				DelayTimer(IN := TRUE);
			END_IF
		ELSE
			DelayTimer(IN := TRUE);
		END_IF
	END_IF

22:	(* wait for scan started *)
	eFwUpdateState := eFwU_ScanningSlaves;

	fbAdsWrite();
	IF NOT fbAdswrite.BUSY THEN
		IF fbAdsWrite.ERR THEN
			IF TestAndSet(bBlockEcatScan) THEN
				IF iBlockEcatScanCount > 0 THEN
					iBlockEcatScanCount := iBlockEcatScanCount - 1;
				END_IF
				bBlockEcatScan := FALSE;
				eFwUpdateState := eFwU_StartScanError;
				bError		:= TRUE;
				iErrId		:= fbAdsWrite.ERRID;
				iAdsErrId	:= UDINT_TO_UINT(iErrId);
				iState		:= 25;
				fbAdsWrite(WRITE:= FALSE);
			END_IF
		ELSE
			iState := iState + 1; (* 23. wait until command is done *)
			fbAdsWrite(WRITE:= FALSE);
		END_IF;
	END_IF;

23: (* wait until command is done *)
	nIdxOffs := SHL(nSDO_IDX_SBP_SCANCOMMANDSTART,16) OR 16#00_00_00_03; (* read reply *)
	fbAdsRead(
		NETID	:= stDriveRef.sNetId,
		PORT	:= EC_AMSPORT_MASTER,
		IDXGRP	:= EC_ADS_IGRP_CANOPEN_SDO,
		IDXOFFS	:= nIdxOffs,
		LEN		:= SIZEOF(stScanStatus),
		DESTADDR:= ADR(stScanStatus),
		READ	:= TRUE,
		TMOUT	:= tTimeout
	);

	IF NOT fbAdsRead.BUSY THEN
		IF fbAdsRead.ERR THEN
			IF TestAndSet(bBlockEcatScan) THEN
				IF iBlockEcatScanCount > 0 THEN
					iBlockEcatScanCount := iBlockEcatScanCount - 1;
				END_IF
				bBlockEcatScan := FALSE;
				eFwUpdateState := eFwU_ScanStateError;
				bError		:= TRUE;
				iErrId		:= fbAdsRead.ERRID;
				iAdsErrId	:= UDINT_TO_UINT(iErrId);
				iState		:= 25;
				fbAdsRead(READ:= FALSE);
			END_IF
		ELSE
			IF 	stScanStatus.nScanStatus = eEcScanSlavesCommandState_Completed_NoErrors_NoReply OR
				stScanStatus.nScanStatus = eEcScanSlavesCommandState_Completed_NoErrors_Reply OR
				stScanStatus.nScanStatus = eEcScanSlavesCommandState_Completed_Error_NoReply OR
				stScanStatus.nScanStatus = eEcScanSlavesCommandState_Completed_Error_Reply
			THEN
				IF stScanStatus.nScanStatus = eEcScanSlavesCommandState_Completed_NoErrors_Reply THEN
					(* 24. get scanned data at found position *)
					nIdxOffs := SHL(nSDO_IDX_SBP_SLAVEINFODATASTART+iSlaveBlockIndex*128+iSlaveIndex-1,16) OR nADSIOFFS_ECAT_COE_COMPLETEACCESS;
					fbAdsRead(READ:= FALSE);
					fbAdsRead(
						NETID	:= stDriveRef.sNetId,
						PORT	:= EC_AMSPORT_MASTER,
						IDXGRP	:= EC_ADS_IGRP_CANOPEN_SDO,
						IDXOFFS	:= nIdxOffs,
						LEN		:= SIZEOF(stLocalInfo),
						DESTADDR:= ADR(stLocalInfo),
						READ	:= TRUE,
						TMOUT	:= tTimeout
					);
					iState := iState + 1;
					fbAdsRead(READ:= FALSE);
				ELSE
					IF TestAndSet(bBlockEcatScan) THEN
						IF iBlockEcatScanCount > 0 THEN
							iBlockEcatScanCount := iBlockEcatScanCount - 1;
						END_IF
						bBlockEcatScan := FALSE;
						eFwUpdateState := eFwU_ScanStateError;
						bError		:= TRUE;
						iErrId		:= 16#719;
						iAdsErrId	:= UDINT_TO_UINT(iErrId);
						iState		:= 25;
						fbAdsRead(READ:= FALSE);
					END_IF
				END_IF;
			ELSE
				iState := iState; (* try it again *)
				fbAdsRead(READ:= FALSE);
			END_IF;
		END_IF;
	END_IF;

24:	(* wait for scanned data *)
	eFwUpdateState := eFwU_ScanningSlaves;

	fbAdsRead();
	IF NOT fbAdsRead.BUSY THEN
		IF TestAndSet(bBlockEcatScan) THEN
			IF iBlockEcatScanCount > 0 THEN
				iBlockEcatScanCount := iBlockEcatScanCount - 1;
			END_IF
			bBlockEcatScan := FALSE;
	
			(*check error and  noOfSlaves > max*)
			IF fbAdsRead.ERR THEN
				eFwUpdateState := eFwU_ScanIdentityError;
				bError		:= TRUE;
				iErrId		:= fbAdsRead.ERRID;
				iAdsErrId	:= UDINT_TO_UINT(iErrId);
				iState		:= 25;
			ELSE
				sScannedType:= F_ConvProductCodeToString(stLocalInfo.stSlaveIdentity);

				IF (LEFT(sScannedType, 3) <> 'AX5') THEN
					(* scanned slave type <> AX5xxx *)
					eFwUpdateState := eFwU_ScannedTypeInNoAX5xxx;
					bError		:= TRUE;
					iErrId		:= 16#70E;
					iAdsErrId	:= UDINT_TO_UINT(iErrId);
					iState		:= 25;
				ELSIF LEFT(sScannedType, 4) <> LEFT(sConfiguredType,4) THEN
					(* mismatch between configured and scanned slave type, e.g. AX52xx <> AX51xx *)
					IF (LEFT(sConfiguredType, 4) = 'AX51') AND (LEFT(sScannedType, 4) = 'AX52') THEN
						eFwUpdateState := eFwU_ChannelMismatch_1Cfg_2Scanned;
					ELSIF(LEFT(sConfiguredType, 4) = 'AX52') AND (LEFT(sScannedType, 4) = 'AX51') THEN
						eFwUpdateState := eFwU_ChannelMismatch_2Cfg_1Scanned;
					ELSIF (LEFT(sConfiguredType, 4) = 'AX50') AND (LEFT(sScannedType, 4) = 'AX51') THEN
						eFwUpdateState := eFwU_ChannelMismatch_0Cfg_1Scanned;
					ELSIF (LEFT(sConfiguredType, 4) = 'AX50') AND (LEFT(sScannedType, 4) = 'AX52') THEN
						eFwUpdateState := eFwU_ChannelMismatch_0Cfg_2Scanned;
					ELSIF (LEFT(sConfiguredType, 4) = 'AX51') AND (LEFT(sScannedType, 4) = 'AX50') THEN
						eFwUpdateState := eFwU_ChannelMismatch_1Cfg_0Scanned;
					ELSIF (LEFT(sConfiguredType, 4) = 'AX52') AND (LEFT(sScannedType, 4) = 'AX50') THEN
						eFwUpdateState := eFwU_ChannelMismatch_2Cfg_0Scanned;
					ELSE
						eFwUpdateState := eFwU_ChannelMismatch;
					END_IF

					bError		:= TRUE;
					iErrId		:= 16#70E;
					iAdsErrId	:= UDINT_TO_UINT(iErrId);
					iState		:= 25;
				ELSIF (MID(sConfiguredType, 2, 5) <> MID(sScannedType, 2, 5)) AND
					(	((LEFT(sConfiguredType, 4) = 'AX51') AND (LEFT(sScannedType, 4) = 'AX51')) OR
						((LEFT(sConfiguredType, 4) = 'AX52') AND (LEFT(sScannedType, 4) = 'AX52'))	) THEN

					bError		:= TRUE;
					iErrId		:= 16#70E;
					iAdsErrId	:= UDINT_TO_UINT(iErrId);
					iState		:= 25;
				ELSE
					(* create firmware file name *)
					sScannedFirmwareFile 	:= '';
					sScannedFirmwareFileDUC := '';
					IF (LEFT(sScannedType, 4) = 'AX50') THEN
						sScannedFirmwareFile := LEFT(sScannedType, 6);								(* --> "AX5021"               *)
						sScannedFirmwareFile := CONCAT(sScannedFirmwareFile, '_xxxx_');				(* --> "AX5021_xxxx_"         *)
					ELSIF (LEFT(sScannedType, 4) = 'AX51') OR (LEFT(sScannedType, 4) = 'AX52') THEN
						sScannedFirmwareFile := 'AX5yxx_xxxx_';									(* --> "AX5yxx_xxxx_"         *)
					END_IF

					sScannedFirmwareFile := CONCAT(sScannedFirmwareFile, RIGHT(sScannedType,4));(* --> "AX5021_xxxx_0002"                 or "AX5yxx_xxxx_0010"   *)
					sScannedFirmwareFile := CONCAT(sScannedFirmwareFile, '_');					(* --> "AX5021_xxxx_0002_"                or "AX5yxx_xxxx_0010_"  *)
					sScannedFirmwareFileDUC := sScannedFirmwareFile;
					sScannedFirmwareFile 	:= F_ToUCase(sScannedFirmwareFile);
					sScannedFirmwareFileDUC	:= F_ToUCase(sScannedFirmwareFileDUC);
					iState := iState + 1;
				END_IF
			END_IF;
			fbAdsRead(READ:= FALSE);
		END_IF
	END_IF;

25:
	IF TestAndSet(bBlockDrivesFwUpdate) THEN
		iArrDrivesUpdatePorts[iNextUpdateIdx] := 0;
		bBlockDrivesFwUpdate := FALSE;

		IF NOT bError THEN
			IF bUpdateViaOtherChn THEN
				eFwUpdateState := eFwU_UpdatedViaOtherChannel;
			ELSE
				eFwUpdateState := eFwU_FwUpdateDone;
			END_IF
		END_IF

		bBusy	:= FALSE;
		iState	:= 0;
	END_IF

END_CASE

bExecute_I := bExecute_I AND bExecute;
END_FUNCTION_BLOCK

(* POU FB_SoEAX5000ReadActMainVoltage_ByDriveRef, ST *)
FUNCTION_BLOCK FB_SoEAX5000ReadActMainVoltage_ByDriveRef
VAR_INPUT
	stDriveRef			: ST_DriveRef; 	(* contains sNetID of EcMaster, nSlaveAddr of EcDrive, nDriveNo of EcDrive, either preset or read from NC *)
	bExecute			: BOOL;			(* Function block execution is triggered by a rising edge at this input.*)
	tTimeout			: TIME := DEFAULT_ADS_TIMEOUT;(* States the time before the function is cancelled. *)
END_VAR
VAR_OUTPUT
	bBusy				: BOOL;
	bError				: BOOL;
	iAdsErrId			: UINT;
	iSercosErrId		: UINT;
	dwAttribute			: DWORD;
	fActualMainVoltage	: REAL;
END_VAR
{library private}
VAR
	fbEcSoERead 		: FB_EcSoERead;
	iState				: INT;
	bExecute_I			: BOOL;
	iErrId				: UDINT;
	iActualMainVoltage	: DINT;
	uiActualMainVoltage	: UDINT;
	dwData				: ARRAY [0..1] OF DWORD;
	cbBufLen			: UDINT;	(* Contains the max. number of bytes to be received. *)

	nFactor				: UINT;					(* bits  0..15 *)
	eLength				: E_SoE_AttribLen;		(* bits 16..18 *)
	eType				: E_SoE_Type;			(* bits 20..22 *)
	nComma				: USINT;				(* bits 24..27 *)
END_VAR
CASE iState OF
0: (* idle *)
	IF bExecute AND NOT bExecute_I THEN
		bExecute_I := bExecute;
		cbBufLen := SIZEOF(dwAttribute) + 2;

		(* read actual main voltage *)
		fbEcSoERead(
			sNetId		:= stDriveRef.sNetId,
			nSlaveAddr	:= stDriveRef.nSlaveAddr,
			nIdn		:= 16#8000 + 200,
			nElement	:= 16#44,
			nDriveNo	:= stDriveRef.nDriveNo,
			bCommand	:= FALSE,
			pDstBuf		:= ADR(dwData),
			cbBufLen	:= SIZEOF(dwData),
			bExecute	:= FALSE,
			tTimeout	:= tTimeout
		);
		fbEcSoERead(bExecute := TRUE);

		iState	:= 10;
		bBusy	:= TRUE;
		bError	:= FALSE;
		iErrId	:= 0;
		iAdsErrId		:= 0;
		iSercosErrId	:= 0;
	END_IF

10: (* wait for read actual main voltage done *)
	fbEcSoERead(bExecute := FALSE);

	IF NOT fbEcSoERead.bBusy THEN
		fbEcSoERead(bExecute := FALSE);
		iState	:= 0;

		IF NOT fbEcSoERead.bError THEN
			bBusy	:= FALSE;
			dwAttribute := dwData[0];
			IF (dwAttribute <> 0) THEN
				nFactor	:= DWORD_TO_UINT(dwAttribute          AND 16#0000FFFF); (* bits  0..15 *)
				eLength	:= DWORD_TO_INT(SHR(dwAttribute,  16) AND 16#00000007);	(* bits 16..18 *)
				eType	:= DWORD_TO_INT(SHR(dwAttribute,  20) AND 16#00000007);	(* bits 20..22 *)
				nComma	:= DWORD_TO_USINT(SHR(dwAttribute,24) AND 16#0000000F); (* bits 24..27 *)
			END_IF

			CASE eType OF
			eSoE_Type_UNSIGNED, eSoE_Type_BIN, eSoE_Type_HEX:
				CASE eLength OF
					eSoE_LEN_2BYTE:
						uiActualMainVoltage := 0;
						MEMCPY(ADR(uiActualMainVoltage), ADR(dwData[1]), UDINT#2);
						fActualMainVoltage := UDINT_TO_REAL(uiActualMainVoltage) * nFactor / EXPT(10,nComma);
					eSoE_LEN_4BYTE:
						MEMCPY(ADR(uiActualMainVoltage), ADR(dwData[1]), UDINT#4);
						fActualMainVoltage := UDINT_TO_REAL(uiActualMainVoltage) * nFactor / EXPT(10,nComma);
					ELSE
						bError := TRUE;
						iErrId := 16#705; (* parameter size not correct *)
						fActualMainVoltage := 0;
				END_CASE

			eSoE_Type_SIGNED:
				CASE eLength OF
					eSoE_LEN_2BYTE:
						iActualMainVoltage := 0;
						MEMCPY(ADR(iActualMainVoltage), ADR(dwData[1]), UDINT#2);
						fActualMainVoltage := DINT_TO_REAL(iActualMainVoltage) * nFactor / EXPT(10,nComma);
					eSoE_LEN_4BYTE:
						MEMCPY(ADR(iActualMainVoltage), ADR(dwData[1]), UDINT#4);
						fActualMainVoltage := DINT_TO_REAL(iActualMainVoltage) * nFactor / EXPT(10,nComma);
					ELSE
						bError := TRUE;
						iErrId := 16#705; (* parameter size not correct *)
						fActualMainVoltage := 0;
				END_CASE

			ELSE
				bError := TRUE;
				iErrId := 16#706; (* invalid parameter value(s) *)
				fActualMainVoltage := 0;
			END_CASE

		ELSE
			bBusy	:= FALSE;
			bError	:= TRUE;
			iErrId	:= fbEcSoERead.nErrId;
			iAdsErrId		:= UDINT_TO_UINT(iErrId);
			iSercosErrId	:= DWORD_TO_UINT(SHR((UDINT_TO_DWORD(iErrId) AND 16#FFFF0000),16));
			fActualMainVoltage := 0;
		END_IF
	END_IF

END_CASE

bExecute_I := bExecute_I AND bExecute;
END_FUNCTION_BLOCK

(* POU FB_SoEAX5000SetMotorCtrlWord_ByDriveRef, ST *)
FUNCTION_BLOCK FB_SoEAX5000SetMotorCtrlWord_ByDriveRef
VAR_INPUT
	stDriveRef		: ST_DriveRef; 	(* contains sNetID of EcMaster, nSlaveAddr of EcDrive, nDriveNo of EcDrive, either preset or read from NC *)
	bExecute		: BOOL;				(* Function block execution is triggered by a rising edge at this input.*)
	tTimeout		: TIME := DEFAULT_ADS_TIMEOUT;(* States the time before the function is cancelled. *)
	bForceLock		: BOOL;
	bForceUnlock	: BOOL;
END_VAR
VAR_OUTPUT
	bBusy			: BOOL;
	bError			: BOOL;
	iAdsErrId		: UINT;
	iSercosErrId	: UINT;
END_VAR
{library private}
VAR
	fbEcSoEWrite 	: FB_EcSoEWrite;
	iState			: INT;
	bExecute_I		: BOOL;
	iMotorCtrlWord	: WORD;
	iErrId			: UDINT;
END_VAR
CASE iState OF
0: (* idle *)
	IF bExecute AND NOT bExecute_I THEN
		bExecute_I := bExecute;

		iMotorCtrlWord.0 := bForceLock;
		iMotorCtrlWord.1 := bForceUnlock;

		(* set Motor Control Word *)
		fbEcSoEWrite(
			sNetId		:= stDriveRef.sNetId,
			nSlaveAddr	:= stDriveRef.nSlaveAddr,
			nIdn		:= 16#8000 + 96,
			nElement	:= 16#40,
			nDriveNo	:= stDriveRef.nDriveNo,
			bCommand	:= FALSE,
			pSrcBuf		:= ADR(iMotorCtrlWord),
			cbBufLen	:= SIZEOF(iMotorCtrlWord),
			bExecute	:= FALSE,
			tTimeout	:= tTimeout
		);
		fbEcSoEWrite(bExecute := TRUE);

		iState	:= 10;
		bBusy	:= TRUE;
		bError	:= FALSE;
		iErrId	:= 0;
		iAdsErrId		:= 0;
		iSercosErrId	:= 0;
	END_IF

10: (* wait for set Motor Control Word done *)
	fbEcSoEWrite(bExecute := FALSE);

	IF NOT fbEcSoEWrite.bBusy THEN
		fbEcSoEWrite(bExecute := FALSE);
		iState	:= 0;

		IF NOT fbEcSoEWrite.bError THEN
			bBusy	:= FALSE;
		ELSE
			bBusy	:= FALSE;
			bError	:= TRUE;
			iErrId	:= fbEcSoEWrite.nErrId;
			iAdsErrId		:= UDINT_TO_UINT(iErrId);
			iSercosErrId	:= DWORD_TO_UINT(SHR((UDINT_TO_DWORD(iErrId) AND 16#FFFF0000),16));
		END_IF
	END_IF

END_CASE

bExecute_I := bExecute_I AND bExecute;
END_FUNCTION_BLOCK

(* POU FB_SoEExecuteCommand_ByDriveRef, ST *)
FUNCTION_BLOCK FB_SoEExecuteCommand_ByDriveRef
(* The  FB_EcSoEWrite sends a SoE write request to an EtherCAT slave device.*)
VAR_INPUT
	stDriveRef		: ST_DriveRef; 	(* contains sNetID of EcMaster, nSlaveAddr of EcDrive, nDriveNo of EcDrive, either preset or read from NC *)
	nIdn			: WORD;			(* SoE IDN: e.g. "S_0_IDN + 1" for S-0-0001 or "P_0_IDN + 23" for P-0-0023*)
	bExecute		: BOOL;			(* Function block execution is triggered by a rising edge at this input.*)
	tTimeout		: TIME := DEFAULT_ADS_TIMEOUT;(* States the time before the function is cancelled. *)
END_VAR
VAR_OUTPUT
	bBusy			: BOOL;
	bError			: BOOL;
	iAdsErrId		: UINT;
	iSercosErrId	: UINT;
END_VAR
{library private}
VAR
	fbEcSoEWrite	: FB_EcSoEWrite;
	iErrId			: UDINT;
	iState			: INT;
	bExecute_I		: BOOL;

	eExecuteCmd		: E_SoE_CmdControl := eSoE_CmdControl_SetAndEnable;
	eCancelCmd		: E_SoE_CmdControl := eSoE_CmdControl_Cancel;
END_VAR
CASE iState OF
0: (* idle *)
	IF bExecute AND NOT bExecute_I THEN
		bExecute_I := bExecute;

		(* execute cmd *)
		fbEcSoEWrite(
			sNetId		:= stDriveRef.sNetId,
			nSlaveAddr	:= stDriveRef.nSlaveAddr,
			nIdn			:= nIdn,
			nElement	:= EC_SOE_ELEMENT_VALUE,
			nDriveNo	:= stDriveRef.nDriveNo,
			bCommand	:= TRUE,
			pSrcBuf		:= ADR(eExecuteCmd),
			cbBufLen	:= SIZEOF(eExecuteCmd),
			bExecute	:= FALSE,
			tTimeout		:= tTimeout
		);
		fbEcSoEWrite(bExecute := TRUE);

		iState	:= 10;
		bBusy	:= TRUE;
		bError	:= FALSE;
		iErrId	:= 0;
		iAdsErrId		:= 0;
		iSercosErrId	:= 0;
	END_IF

10: (* wait for execute  done *)
	fbEcSoEWrite(bExecute := FALSE);

	IF NOT fbEcSoEWrite.bBusy THEN
		fbEcSoEWrite(bExecute := FALSE);

		iState	:= 0;
		bBusy	:= FALSE;

		IF fbEcSoEWrite.bError THEN
			bError	:= TRUE;
			iErrId	:= fbEcSoEWrite.nErrId;
			iAdsErrId		:= UDINT_TO_UINT(iErrId);
			iSercosErrId	:= DWORD_TO_UINT(SHR((UDINT_TO_DWORD(iErrId) AND 16#FFFF0000),16));
		END_IF
	END_IF
END_CASE

bExecute_I := bExecute_I AND bExecute;
END_FUNCTION_BLOCK

(* POU FB_SoEReadAmplifierTemperature_ByDriveRef, ST *)
FUNCTION_BLOCK FB_SoEReadAmplifierTemperature_ByDriveRef
VAR_INPUT
	stDriveRef				: ST_DriveRef; 	(* contains sNetID of EcMaster, nSlaveAddr of EcDrive, nDriveNo of EcDrive, either preset or read from NC *)
	bExecute				: BOOL;				(* Function block execution is triggered by a rising edge at this input.*)
	tTimeout				: TIME := DEFAULT_ADS_TIMEOUT;(* States the time before the function is cancelled. *)
END_VAR
VAR_OUTPUT
	bBusy					: BOOL;
	bError					: BOOL;
	iAdsErrId				: UINT;
	iSercosErrId			: UINT;
	dwAttribute				: DWORD;
	fAmplifierTemperature	: REAL;
END_VAR
{library private}
VAR
	fbEcSoERead 			: FB_EcSoERead;
	iState					: INT;
	bExecute_I				: BOOL;
	iErrId					: UDINT;
	iAmplifierTemperature	: DINT;
	uiAmplifierTemperature	: UDINT;
	dwData					: ARRAY [0..1] OF DWORD;

	nFactor				: UINT;					(* bits  0..15 *)
	eLength				: E_SoE_AttribLen;		(* bits 16..18 *)
	eType				: E_SoE_Type;			(* bits 20..22 *)
	nComma				: USINT;				(* bits 24..27 *)
END_VAR
CASE iState OF
0: (* idle *)
	IF bExecute AND NOT bExecute_I THEN
		bExecute_I := bExecute;

		IF NOT bSeqReadDrvAttrAndValue THEN
			(* read Amplifier Temperature *)
			fbEcSoERead(
				sNetId		:= stDriveRef.sNetId,
				nSlaveAddr	:= stDriveRef.nSlaveAddr,
				nIdn		:= 384,
				nElement	:= 16#44, (* EC_SOE_ELEMENT_VALUE | EC_SOE_ELEMENT_ATTRIBUTE *)
				nDriveNo	:= stDriveRef.nDriveNo,
				bCommand	:= FALSE,
				pDstBuf		:= ADR(dwData),
				cbBufLen	:= SIZEOF(dwData),
				bExecute	:= FALSE,
				tTimeout	:= tTimeout
			);
			iState	:= 10;
		ELSE
			(* read attribute and Amplifier Temperature sequentially *)
			fbEcSoERead(
				sNetId		:= stDriveRef.sNetId,
				nSlaveAddr	:= stDriveRef.nSlaveAddr,
				nIdn		:= 384,
				nElement	:= EC_SOE_ELEMENT_ATTRIBUTE,
				nDriveNo	:= stDriveRef.nDriveNo,
				bCommand	:= FALSE,
				pDstBuf		:= ADR(dwData[0]),
				cbBufLen	:= SIZEOF(dwData[0]),
				bExecute	:= FALSE,
				tTimeout	:= tTimeout
			);
			iState	:= 5;
		END_IF
		fbEcSoERead(bExecute := TRUE);

		bBusy	:= TRUE;
		bError	:= FALSE;
		iErrId	:= 0;
		iAdsErrId		:= 0;
		iSercosErrId	:= 0;
	END_IF

5: (* wait for read Amplifier Temperature done *)
	fbEcSoERead(bExecute := FALSE);

	IF NOT fbEcSoERead.bBusy THEN
		fbEcSoERead(bExecute := FALSE);

		IF NOT fbEcSoERead.bError THEN
			(* read attribute and Amplifier Temperature sequentially *)
			fbEcSoERead(
				sNetId		:= stDriveRef.sNetId,
				nSlaveAddr	:= stDriveRef.nSlaveAddr,
				nIdn		:= 384,
				nElement	:= EC_SOE_ELEMENT_VALUE,
				nDriveNo	:= stDriveRef.nDriveNo,
				bCommand	:= FALSE,
				pDstBuf		:= ADR(dwData[1]),
				cbBufLen	:= SIZEOF(dwData[1]),
				bExecute	:= FALSE,
				tTimeout	:= tTimeout
			);
			fbEcSoERead(bExecute := TRUE);
			iState	:= 10;
		ELSE
			bBusy	:= FALSE;
			bError	:= TRUE;
			iErrId	:= fbEcSoERead.nErrId;
			iAdsErrId		:= UDINT_TO_UINT(iErrId);
			iSercosErrId	:= DWORD_TO_UINT(SHR((UDINT_TO_DWORD(iErrId) AND 16#FFFF0000),16));
			fAmplifierTemperature := 0;
			iState	:= 0;
		END_IF
	END_IF

10: (* wait for read Amplifier Temperature done *)
	fbEcSoERead(bExecute := FALSE);

	IF NOT fbEcSoERead.bBusy THEN
		fbEcSoERead(bExecute := FALSE);
		iState	:= 0;

		IF NOT fbEcSoERead.bError THEN
			bBusy	:= FALSE;
			dwAttribute := dwData[0];
			IF (dwAttribute <> 0) THEN
				nFactor	:= DWORD_TO_UINT(dwAttribute          AND 16#0000FFFF); (* bits  0..15 *)
				eLength	:= DWORD_TO_INT(SHR(dwAttribute,  16) AND 16#00000007);	(* bits 16..18 *)
				eType	:= DWORD_TO_INT(SHR(dwAttribute,  20) AND 16#00000007);	(* bits 20..22 *)
				nComma	:= DWORD_TO_USINT(SHR(dwAttribute,24) AND 16#0000000F); (* bits 24..27 *)
			END_IF

			CASE eType OF
			eSoE_Type_UNSIGNED, eSoE_Type_BIN, eSoE_Type_HEX:
				CASE eLength OF
					eSoE_LEN_2BYTE:
						uiAmplifierTemperature := 0;
						MEMCPY(ADR(uiAmplifierTemperature), ADR(dwData[1]), UDINT#2);
						fAmplifierTemperature := UDINT_TO_REAL(uiAmplifierTemperature) * nFactor / EXPT(10,nComma);
					eSoE_LEN_4BYTE:
						MEMCPY(ADR(uiAmplifierTemperature), ADR(dwData[1]), UDINT#4);
						fAmplifierTemperature := UDINT_TO_REAL(uiAmplifierTemperature) * nFactor / EXPT(10,nComma);
					ELSE
						bError := TRUE;
						iErrId := 16#705; (* parameter size not correct *)
						fAmplifierTemperature := 0;
				END_CASE

			eSoE_Type_SIGNED:
				CASE eLength OF
					eSoE_LEN_2BYTE:
						iAmplifierTemperature := 0;
						MEMCPY(ADR(iAmplifierTemperature), ADR(dwData[1]), UDINT#2);
						fAmplifierTemperature := DINT_TO_REAL(iAmplifierTemperature) * nFactor / EXPT(10,nComma);
					eSoE_LEN_4BYTE:
						MEMCPY(ADR(iAmplifierTemperature), ADR(dwData[1]), UDINT#4);
						fAmplifierTemperature := DINT_TO_REAL(iAmplifierTemperature) * nFactor / EXPT(10,nComma);
					ELSE
						bError := TRUE;
						iErrId := 16#705; (* parameter size not correct *)
						fAmplifierTemperature := 0;
				END_CASE

			ELSE
				bError := TRUE;
				iErrId := 16#706; (* invalid parameter value(s) *)
				fAmplifierTemperature := 0;
			END_CASE

		ELSE
			bBusy	:= FALSE;
			bError	:= TRUE;
			iErrId	:= fbEcSoERead.nErrId;
			iAdsErrId		:= UDINT_TO_UINT(iErrId);
			iSercosErrId	:= DWORD_TO_UINT(SHR((UDINT_TO_DWORD(iErrId) AND 16#FFFF0000),16));
			fAmplifierTemperature := 0;
		END_IF
	END_IF

END_CASE

bExecute_I := bExecute_I AND bExecute;
END_FUNCTION_BLOCK

(* POU FB_SoEReadClassXDiag_ByDriveRef, ST *)
FUNCTION_BLOCK FB_SoEReadClassXDiag_ByDriveRef
VAR_INPUT
	stDriveRef		: ST_DriveRef; 	(* contains sNetID of EcMaster, nSlaveAddr of EcDrive, nDriveNo of EcDrive, either preset or read from NC *)
	bExecute		: BOOL;			(* Function block execution is triggered by a rising edge at this input.*)
	iDiagClass		: USINT:= 1;	(* 1: C1D (S-0-0011) is default, 2: C2D (S-0-0012), 3: C3D (S-0-0013) *)
	tTimeout		: TIME := DEFAULT_ADS_TIMEOUT;(* States the time before the function is cancelled. *)
END_VAR
VAR_OUTPUT
	bBusy			: BOOL;
	bError			: BOOL;
	iAdsErrId		: UINT;
	iSercosErrId	: UINT;
	dwAttribute		: DWORD;
	wClassXDiag		: WORD;
END_VAR
{library private}
VAR
	fbEcSoERead 	: FB_EcSoERead;
	iState			: INT;
	bExecute_I		: BOOL;
	iErrId			: UDINT;
	dwData			: ARRAY [0..1] OF DWORD;
	iSParamNum		: WORD;

	nFactor			: UINT;					(* bits  0..15 *)
	eLength			: E_SoE_AttribLen;		(* bits 16..18 *)
	eType			: E_SoE_Type;			(* bits 20..22 *)
	nComma			: USINT;				(* bits 24..27 *)
END_VAR
CASE iState OF
0: (* idle *)
	IF bExecute AND NOT bExecute_I THEN
		bExecute_I := bExecute;

		CASE iDiagClass OF
		1:	iSParamNum := 11; (* C1D *)
		2:	iSParamNum := 12; (* C2D *)
		3:	iSParamNum := 13; (* C3D *)
		ELSE
			iSParamNum := 11; (* C1D *)
		END_CASE

		IF NOT bSeqReadDrvAttrAndValue THEN
			(* read drive diag number *)
			fbEcSoERead(
				sNetId		:= stDriveRef.sNetId,
				nSlaveAddr	:= stDriveRef.nSlaveAddr,
				nIdn		:= iSParamNum,
				nElement	:= 16#44, (* EC_SOE_ELEMENT_VALUE | EC_SOE_ELEMENT_ATTRIBUTE *)
				nDriveNo	:= stDriveRef.nDriveNo,
				bCommand	:= FALSE,
				pDstBuf		:= ADR(dwData),
				cbBufLen	:= SIZEOF(dwData),
				bExecute	:= FALSE,
				tTimeout	:= tTimeout
			);
			iState	:= 10;
		ELSE
			(* read attribute and drive diag number sequentially *)
			fbEcSoERead(
				sNetId		:= stDriveRef.sNetId,
				nSlaveAddr	:= stDriveRef.nSlaveAddr,
				nIdn		:= iSParamNum,
				nElement	:= EC_SOE_ELEMENT_ATTRIBUTE,
				nDriveNo	:= stDriveRef.nDriveNo,
				bCommand	:= FALSE,
				pDstBuf		:= ADR(dwData[0]),
				cbBufLen	:= SIZEOF(dwData[0]),
				bExecute	:= FALSE,
				tTimeout	:= tTimeout
			);
			iState	:= 5;
		END_IF
		fbEcSoERead(bExecute := TRUE);

		bBusy	:= TRUE;
		bError	:= FALSE;
		iErrId	:= 0;
		iAdsErrId		:= 0;
		iSercosErrId	:= 0;
	END_IF

5:	(* read attribute and drive diag number sequentially *)
	fbEcSoERead(bExecute := FALSE);

	IF NOT fbEcSoERead.bBusy THEN
		fbEcSoERead(bExecute := FALSE);

		IF NOT fbEcSoERead.bError THEN
			fbEcSoERead(
				sNetId		:= stDriveRef.sNetId,
				nSlaveAddr	:= stDriveRef.nSlaveAddr,
				nIdn		:= iSParamNum,
				nElement	:= EC_SOE_ELEMENT_VALUE,
				nDriveNo	:= stDriveRef.nDriveNo,
				bCommand	:= FALSE,
				pDstBuf		:= ADR(dwData[1]),
				cbBufLen	:= SIZEOF(dwData[1]),
				bExecute	:= FALSE,
				tTimeout	:= tTimeout
			);
			fbEcSoERead(bExecute := TRUE);
			iState	:= 10;

		ELSE
			bBusy	:= FALSE;
			bError	:= TRUE;
			iErrId	:= fbEcSoERead.nErrId;
			iAdsErrId		:= UDINT_TO_UINT(iErrId);
			iSercosErrId	:= DWORD_TO_UINT(SHR((UDINT_TO_DWORD(iErrId) AND 16#FFFF0000),16));
			wClassXDiag := 0;
			iState	:= 0;
		END_IF
	END_IF

10: (* wait for read drive diag done *)
	fbEcSoERead(bExecute := FALSE);

	IF NOT fbEcSoERead.bBusy THEN
		fbEcSoERead(bExecute := FALSE);
		iState	:= 0;

		IF NOT fbEcSoERead.bError THEN
			bBusy	:= FALSE;
			dwAttribute := dwData[0];
			IF (dwAttribute <> 0) THEN
				nFactor	:= DWORD_TO_UINT(dwAttribute          AND 16#0000FFFF); (* bits  0..15 *)
				eLength	:= DWORD_TO_INT(SHR(dwAttribute,  16) AND 16#00000007);	(* bits 16..18 *)
				eType	:= DWORD_TO_INT(SHR(dwAttribute,  20) AND 16#00000007);	(* bits 20..22 *)
				nComma	:= DWORD_TO_USINT(SHR(dwAttribute,24) AND 16#0000000F); (* bits 24..27 *)
			END_IF

			CASE eType OF
			eSoE_Type_UNSIGNED, eSoE_Type_BIN, eSoE_Type_HEX:
				CASE eLength OF
					eSoE_LEN_2BYTE:
						wClassXDiag := 0;
						MEMCPY(ADR(wClassXDiag), ADR(dwData[1]), UDINT#2);
					ELSE
						bError := TRUE;
						iErrId := 16#705; (* parameter size not correct *)
						wClassXDiag := 0;
				END_CASE

			eSoE_Type_SIGNED:
				CASE eLength OF
					eSoE_LEN_2BYTE:
						wClassXDiag := 0;
						MEMCPY(ADR(wClassXDiag), ADR(dwData[1]), UDINT#2);
					ELSE
						bError := TRUE;
						iErrId := 16#705; (* parameter size not correct *)
						wClassXDiag := 0;
				END_CASE

			ELSE
				bError := TRUE;
				iErrId := 16#706; (* invalid parameter value(s) *)
				wClassXDiag := 0;
			END_CASE
		ELSE
			bBusy	:= FALSE;
			bError	:= TRUE;
			iErrId	:= fbEcSoERead.nErrId;
			iAdsErrId		:= UDINT_TO_UINT(iErrId);
			iSercosErrId	:= DWORD_TO_UINT(SHR((UDINT_TO_DWORD(iErrId) AND 16#FFFF0000),16));
			wClassXDiag := 0;
		END_IF
	END_IF

END_CASE

bExecute_I := bExecute_I AND bExecute;
END_FUNCTION_BLOCK

(* POU FB_SoEReadCommandState_ByDriveRef, ST *)
FUNCTION_BLOCK FB_SoEReadCommandState_ByDriveRef
(* The   FB_EcSoERead sends a SoE read request to an EtherCAT slave device.*)
VAR_INPUT
	stDriveRef		: ST_DriveRef; 	(* contains sNetID of EcMaster, nSlaveAddr of EcDrive, nDriveNo of EcDrive, either preset or read from NC *)
	nIdn			: WORD;		(* SoE IDN: e.g. "S_0_IDN + 1" for S-0-0001 or "P_0_IDN + 23" for P-0-0023*)
	bExecute		: BOOL;		(* Function block execution is triggered by a rising edge at this input.*)
	tTimeout		: TIME := DEFAULT_ADS_TIMEOUT;(* States the time before the function is cancelled. *)
END_VAR
VAR_OUTPUT
	bBusy			: BOOL;
	bError			: BOOL;
	eCmdState		: E_SoE_CmdState;
	iAdsErrId		: UINT;
	iSercosErrId	: UINT;
END_VAR
{library private}
VAR
	fbEcSoERead		: FB_EcSoERead;
	iState			: INT;
	bExecute_I		: BOOL;
	iErrId			: UDINT;
	dwData			: ARRAY [0..1] OF DWORD;
END_VAR
CASE iState OF
0: (* idle *)
	IF bExecute AND NOT bExecute_I THEN
		bExecute_I := bExecute;

		(* read command state *)
		fbEcSoERead(
			sNetId		:= stDriveRef.sNetId,
			nSlaveAddr	:= stDriveRef.nSlaveAddr,
			nIdn		:= nIdn,
			nElement	:= EC_SOE_ELEMENT_DATASTATE,
			nDriveNo	:= stDriveRef.nDriveNo,
			bCommand	:= FALSE,
			pDstBuf		:= ADR(eCmdState),
			cbBufLen	:= SIZEOF(eCmdState),
			bExecute	:= FALSE,
			tTimeout	:= tTimeout
		);
		fbEcSoERead(bExecute := TRUE);

		iState	:= 20;

		bBusy	:= TRUE;
		bError	:= FALSE;
		iErrId	:= 0;
		iAdsErrId		:= 0;
		iSercosErrId	:= 0;
	END_IF


20: (* wait for read ata done *)
	fbEcSoERead(bExecute := FALSE);

	IF NOT fbEcSoERead.bBusy THEN
		fbEcSoERead(bExecute := FALSE);
		iState			:= 0;

		IF NOT fbEcSoERead.bError THEN
			bBusy	:= FALSE;
		ELSE
			bBusy	:= FALSE;
			bError	:= TRUE;
			iErrId	:= fbEcSoERead.nErrId;
			iAdsErrId		:= UDINT_TO_UINT(iErrId);
			iSercosErrId	:= DWORD_TO_UINT(SHR((UDINT_TO_DWORD(iErrId) AND 16#FFFF0000),16));
		END_IF
	END_IF

END_CASE

bExecute_I := bExecute_I AND bExecute;
END_FUNCTION_BLOCK

(* POU FB_SoEReadDcBusCurrent_ByDriveRef, ST *)
FUNCTION_BLOCK FB_SoEReadDcBusCurrent_ByDriveRef
VAR_INPUT
	stDriveRef		: ST_DriveRef; 	(* contains sNetID of EcMaster, nSlaveAddr of EcDrive, nDriveNo of EcDrive, either preset or read from NC *)
	bExecute		: BOOL;			(* Function block execution is triggered by a rising edge at this input.*)
	tTimeout		: TIME := DEFAULT_ADS_TIMEOUT;(* States the time before the function is cancelled. *)
END_VAR
VAR_OUTPUT
	bBusy			: BOOL;
	bError			: BOOL;
	iAdsErrId		: UINT;
	iSercosErrId	: UINT;
	dwAttribute		: DWORD;
	fDcBusCurrent	: REAL;
END_VAR
{library private}
VAR
	fbEcSoERead 	: FB_EcSoERead;
	iState			: INT;
	bExecute_I		: BOOL;
	iErrId			: UDINT;
	iDcBusCurrent	: DINT;
	uiDcBusCurrent	: UDINT;
	dwData			: ARRAY [0..1] OF DWORD;

	nFactor			: UINT;					(* bits  0..15 *)
	eLength			: E_SoE_AttribLen;		(* bits 16..18 *)
	eType			: E_SoE_Type;			(* bits 20..22 *)
	nComma			: USINT;				(* bits 24..27 *)
END_VAR
CASE iState OF
0: (* idle *)
	IF bExecute AND NOT bExecute_I THEN
		bExecute_I := bExecute;

		IF NOT bSeqReadDrvAttrAndValue THEN
			(* read DC bus current *)
			fbEcSoERead(
				sNetId		:= stDriveRef.sNetId,
				nSlaveAddr	:= stDriveRef.nSlaveAddr,
				nIdn		:= 381,
				nElement	:= 16#44, (* EC_SOE_ELEMENT_VALUE | EC_SOE_ELEMENT_ATTRIBUTE *)
				nDriveNo	:= stDriveRef.nDriveNo,
				bCommand	:= FALSE,
				pDstBuf		:= ADR(dwData),
				cbBufLen	:= SIZEOF(dwData),
				bExecute	:= FALSE,
				tTimeout	:= tTimeout
			);
			iState	:= 10;
		ELSE
			(* read attribute and DC bus current sequentially *)
			fbEcSoERead(
				sNetId		:= stDriveRef.sNetId,
				nSlaveAddr	:= stDriveRef.nSlaveAddr,
				nIdn		:= 381,
				nElement	:= EC_SOE_ELEMENT_ATTRIBUTE,
				nDriveNo	:= stDriveRef.nDriveNo,
				bCommand	:= FALSE,
				pDstBuf		:= ADR(dwData[0]),
				cbBufLen	:= SIZEOF(dwData[0]),
				bExecute	:= FALSE,
				tTimeout	:= tTimeout
			);
			iState	:= 5;
		END_IF
		fbEcSoERead(bExecute := TRUE);

		bBusy	:= TRUE;
		bError	:= FALSE;
		iErrId	:= 0;
		iAdsErrId		:= 0;
		iSercosErrId	:= 0;
	END_IF

5: (* wait for read DC bus current done *)
	fbEcSoERead(bExecute := FALSE);

	IF NOT fbEcSoERead.bBusy THEN
		fbEcSoERead(bExecute := FALSE);

		IF NOT fbEcSoERead.bError THEN
			(* read attribute and DC bus current sequentially *)
			fbEcSoERead(
				sNetId		:= stDriveRef.sNetId,
				nSlaveAddr	:= stDriveRef.nSlaveAddr,
				nIdn		:= 381,
				nElement	:= EC_SOE_ELEMENT_VALUE,
				nDriveNo	:= stDriveRef.nDriveNo,
				bCommand	:= FALSE,
				pDstBuf		:= ADR(dwData[1]),
				cbBufLen	:= SIZEOF(dwData[1]),
				bExecute	:= FALSE,
				tTimeout	:= tTimeout
			);
			fbEcSoERead(bExecute := TRUE);
			iState	:= 10;
		ELSE
			bBusy	:= FALSE;
			bError	:= TRUE;
			iErrId	:= fbEcSoERead.nErrId;
			iAdsErrId		:= UDINT_TO_UINT(iErrId);
			iSercosErrId	:= DWORD_TO_UINT(SHR((UDINT_TO_DWORD(iErrId) AND 16#FFFF0000),16));
			fDcBusCurrent := 0;
			iState	:= 0;
		END_IF
	END_IF

10: (* wait for read DC bus current done *)
	fbEcSoERead(bExecute := FALSE);

	IF NOT fbEcSoERead.bBusy THEN
		fbEcSoERead(bExecute := FALSE);
		iState	:= 0;

		IF NOT fbEcSoERead.bError THEN
			bBusy	:= FALSE;
			dwAttribute := dwData[0];
			IF (dwAttribute <> 0) THEN
				nFactor	:= DWORD_TO_UINT(dwAttribute          AND 16#0000FFFF); (* bits  0..15 *)
				eLength	:= DWORD_TO_INT(SHR(dwAttribute,  16) AND 16#00000007);	(* bits 16..18 *)
				eType	:= DWORD_TO_INT(SHR(dwAttribute,  20) AND 16#00000007);	(* bits 20..22 *)
				nComma	:= DWORD_TO_USINT(SHR(dwAttribute,24) AND 16#0000000F); (* bits 24..27 *)
			END_IF

			CASE eType OF
			eSoE_Type_UNSIGNED, eSoE_Type_BIN, eSoE_Type_HEX:
				CASE eLength OF
					eSoE_LEN_2BYTE:
						uiDcBusCurrent := 0;
						MEMCPY(ADR(uiDcBusCurrent), ADR(dwData[1]), UDINT#2);
						fDcBusCurrent := UDINT_TO_REAL(uiDcBusCurrent) * nFactor / EXPT(10,nComma);
					eSoE_LEN_4BYTE:
						MEMCPY(ADR(uiDcBusCurrent), ADR(dwData[1]), UDINT#4);
						fDcBusCurrent := UDINT_TO_REAL(uiDcBusCurrent) * nFactor / EXPT(10,nComma);
					ELSE
						bError := TRUE;
						iErrId := 16#705; (* parameter size not correct *)
						fDcBusCurrent := 0;
				END_CASE

			eSoE_Type_SIGNED:
				CASE eLength OF
					eSoE_LEN_2BYTE:
						iDcBusCurrent := 0;
						MEMCPY(ADR(iDcBusCurrent), ADR(dwData[1]), UDINT#2);
						fDcBusCurrent := DINT_TO_REAL(iDcBusCurrent) * nFactor / EXPT(10,nComma);
					eSoE_LEN_4BYTE:
						MEMCPY(ADR(iDcBusCurrent), ADR(dwData[1]), UDINT#4);
						fDcBusCurrent := DINT_TO_REAL(iDcBusCurrent) * nFactor / EXPT(10,nComma);
					ELSE
						bError := TRUE;
						iErrId := 16#705; (* parameter size not correct *)
						fDcBusCurrent := 0;
				END_CASE

			ELSE
				bError := TRUE;
				iErrId := 16#706; (* invalid parameter value(s) *)
				fDcBusCurrent := 0;
			END_CASE

		ELSE
			bBusy	:= FALSE;
			bError	:= TRUE;
			iErrId	:= fbEcSoERead.nErrId;
			iAdsErrId		:= UDINT_TO_UINT(iErrId);
			iSercosErrId	:= DWORD_TO_UINT(SHR((UDINT_TO_DWORD(iErrId) AND 16#FFFF0000),16));
			fDcBusCurrent := 0;
		END_IF
	END_IF

END_CASE

bExecute_I := bExecute_I AND bExecute;
END_FUNCTION_BLOCK

(* POU FB_SoEReadDcBusVoltage_ByDriveRef, ST *)
FUNCTION_BLOCK FB_SoEReadDcBusVoltage_ByDriveRef
VAR_INPUT
	stDriveRef		: ST_DriveRef; 	(* contains sNetID of EcMaster, nSlaveAddr of EcDrive, nDriveNo of EcDrive, either preset or read from NC *)
	bExecute		: BOOL;			(* Function block execution is triggered by a rising edge at this input.*)
	tTimeout		: TIME := DEFAULT_ADS_TIMEOUT;(* States the time before the function is cancelled. *)
END_VAR
VAR_OUTPUT
	bBusy			: BOOL;
	bError			: BOOL;
	iAdsErrId		: UINT;
	iSercosErrId	: UINT;
	dwAttribute		: DWORD;
	fDcBusVoltage	: REAL;
END_VAR
{library private}
VAR
	fbEcSoERead 	: FB_EcSoERead;
	iState			: INT;
	bExecute_I		: BOOL;
	iErrId			: UDINT;
	iDcBusVoltage	: DINT;
	uiDcBusVoltage	: UDINT;
	dwData			: ARRAY [0..1] OF DWORD;

	nFactor			: UINT;					(* bits  0..15 *)
	eLength			: E_SoE_AttribLen;		(* bits 16..18 *)
	eType			: E_SoE_Type;			(* bits 20..22 *)
	nComma			: USINT;				(* bits 24..27 *)
END_VAR
CASE iState OF
0: (* idle *)
	IF bExecute AND NOT bExecute_I THEN
		bExecute_I := bExecute;

